Yaskawa INFORM job: SUPERDUPLEX_HALFBODY_11_02.JBI

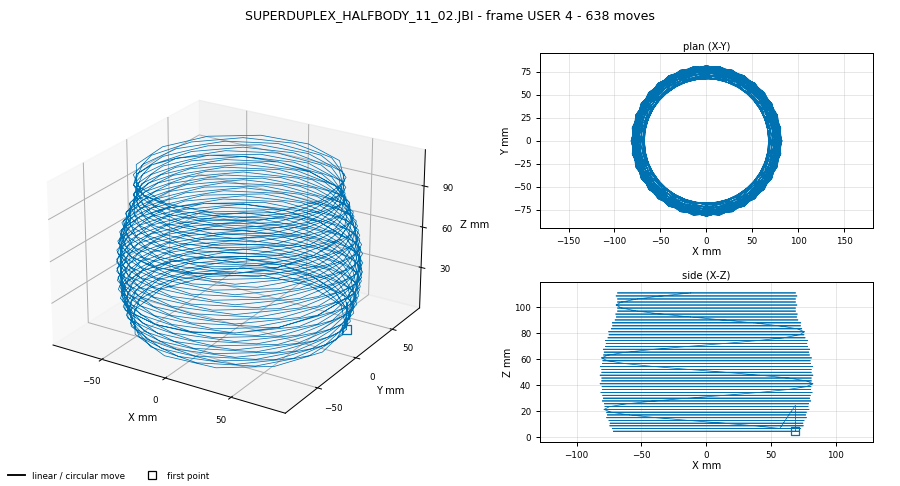
[picture p0: tool path of SUPERDUPLEX_HALFBODY_11_02.JBI in frame USER 4, 638 of 639 moves have a stored position in this frame; points joined in program order, loops and branches not executed]
/JOB
//NAME SUPERDUPLEX_HALFBODY_11_02
///FOLDERNAME SUPERDUPLEX_HALFBODY
//POS
///NPOS 638,0,639,1,0,0
///TOOL 9
///POSTYPE PULSE
P0=8353,-34220,-84194,-128214,7285,517082
///TOOL 9
///USER 4
///POSTYPE USER
///RECTAN
///RCONF 0,0,0,0,0,0,0,0,0,0,0,0,0,0,0,0,0,0,0,0,0,0,0,0
C0=68.785,24.654,4.486,-180.000,-180.000,134.719
C1=72.078,-12.983,4.486,-180.000,180.000,104.834
C2=56.111,-47.225,4.486,-180.000,180.000,74.949
C3=25.162,-68.896,4.486,-180.000,180.000,45.063
C4=-12.476,-72.189,4.486,180.000,180.000,15.136
C5=-46.717,-56.221,4.486,0.000,0.000,165.209
C6=-68.388,-25.273,4.486,0.000,0.000,135.282
C7=-71.681,12.365,4.486,0.000,0.000,105.166
C8=-55.714,46.607,4.486,0.000,0.000,75.051
C9=-24.765,68.278,4.486,0.000,0.000,44.936
C10=12.873,71.570,4.486,0.000,0.000,14.864
C11=47.115,55.603,4.486,-180.000,-180.000,164.791
C12=68.785,24.654,4.486,-180.000,-180.000,134.719
C13=68.785,24.654,24.486,-180.000,-180.000,134.719
C14=56.727,47.124,6.581,160.821,171.291,153.526
C15=25.437,69.033,6.581,-19.179,8.709,3.526
C16=-12.615,72.363,6.581,-19.179,8.709,33.526
C17=-47.234,56.219,6.581,-19.179,8.709,63.526
C18=-69.144,24.930,6.581,-19.179,8.709,93.526
C19=-72.473,-13.123,6.581,-19.179,8.709,123.526
C20=-56.330,-47.742,6.581,-19.179,8.709,153.526
C21=-25.040,-69.651,6.581,160.821,171.291,3.526
C22=13.013,-72.981,6.581,160.821,171.291,33.526
C23=47.632,-56.837,6.581,160.821,171.291,63.526
C24=69.541,-25.548,6.581,160.821,171.291,93.526
C25=72.870,12.505,6.581,160.821,171.291,123.526
C26=56.727,47.124,6.581,160.821,171.291,153.526
C27=37.536,64.360,8.629,158.693,170.383,173.187
C28=64.868,37.028,8.629,158.693,170.383,143.187
C29=74.872,-0.309,8.629,158.693,170.383,113.187
C30=64.868,-37.646,8.629,158.693,170.383,83.187
C31=37.536,-64.978,8.629,158.693,170.383,53.187
C32=0.199,-74.983,8.629,158.693,170.383,23.187
C33=-37.138,-64.978,8.629,-21.307,9.617,173.187
C34=-64.471,-37.646,8.629,-21.307,9.617,143.187
C35=-74.475,-0.309,8.629,-21.307,9.617,113.187
C36=-64.471,37.028,8.629,-21.307,9.617,83.187
C37=-37.138,64.360,8.629,-21.307,9.617,53.187
C38=0.199,74.365,8.629,-21.307,9.617,23.187
C39=37.536,64.360,8.629,158.693,170.383,173.187
C40=13.320,74.103,10.674,-21.438,9.672,13.165
C41=-25.644,70.694,10.674,-21.438,9.672,43.165
C42=-57.683,48.260,10.674,-21.438,9.672,73.165
C43=-74.213,12.812,10.674,-21.438,9.672,103.165
C44=-70.804,-26.152,10.674,-21.438,9.672,133.165
C45=-48.370,-58.191,10.674,-21.438,9.672,163.165
C46=-12.922,-74.721,10.674,158.562,170.328,13.165
C47=26.042,-71.312,10.674,158.562,170.328,43.165
C48=58.081,-48.878,10.674,158.562,170.328,73.165
C49=74.611,-13.430,10.674,158.562,170.328,103.165
C50=71.202,25.534,10.674,158.562,170.328,133.165
C51=48.768,57.573,10.674,158.562,170.328,163.165
C52=13.320,74.103,10.674,-21.438,9.672,13.165
C53=-13.072,74.951,12.739,-20.717,9.367,33.284
C54=26.336,71.504,12.739,-20.717,9.367,3.284
C55=58.741,48.814,12.739,159.283,170.633,153.284
C56=75.459,12.961,12.739,159.283,170.633,123.284
C57=72.012,-26.447,12.739,159.283,170.633,93.284
C58=49.322,-58.851,12.739,159.283,170.633,63.284
C59=13.469,-75.570,12.739,159.283,170.633,33.284
C60=-25.939,-72.122,12.739,159.283,170.633,3.284
C61=-58.344,-49.432,12.739,-20.717,9.367,153.284
C62=-75.062,-13.580,12.739,-20.717,9.367,123.284
C63=-71.614,25.829,12.739,-20.717,9.367,93.284
C64=-48.924,58.233,12.739,-20.717,9.367,63.284
C65=-13.072,74.951,12.739,-20.717,9.367,33.284
C66=-38.329,66.423,14.886,-14.976,6.871,54.096
C67=-66.533,38.219,14.886,-14.976,6.871,84.096
C68=-76.856,-0.309,14.886,-14.976,6.871,114.096
C69=-66.533,-38.837,14.886,-14.976,6.871,144.096
C70=-38.329,-67.041,14.886,-14.976,6.871,174.096
C71=0.199,-77.364,14.886,165.024,173.129,24.096
C72=38.726,-67.041,14.886,165.024,173.129,54.096
C73=66.931,-38.837,14.886,165.024,173.129,84.096
C74=77.254,-0.309,14.886,165.024,173.129,114.096
C75=66.931,38.219,14.886,165.024,173.129,144.096
C76=38.726,66.423,14.886,165.024,173.129,174.096
C77=0.199,76.746,14.886,-14.976,6.871,24.096
C78=-38.329,66.423,14.886,-14.976,6.871,54.096
C79=-59.325,49.637,17.023,-15.358,7.041,74.050
C80=-26.377,72.708,17.023,-15.358,7.041,44.050
C81=13.692,76.213,17.023,-15.358,7.041,14.050
C82=50.145,59.215,17.023,164.642,172.959,164.050
C83=73.216,26.267,17.023,164.642,172.959,134.050
C84=76.721,-13.802,17.023,164.642,172.959,104.050
C85=59.723,-50.256,17.023,164.642,172.959,74.049
C86=26.775,-73.326,17.023,164.642,172.959,44.050
C87=-13.294,-76.831,17.023,164.642,172.959,14.050
C88=-49.748,-59.833,17.023,-15.358,7.041,164.050
C89=-72.818,-26.885,17.023,-15.358,7.041,134.050
C90=-76.324,13.184,17.023,-15.358,7.041,104.050
C91=-59.325,49.637,17.023,-15.358,7.041,74.050
C92=-73.436,26.492,19.138,-15.733,7.206,94.003
C93=-76.971,-13.916,19.138,-15.733,7.206,124.003
C94=-59.829,-50.678,19.138,-15.733,7.206,154.003
C95=-26.602,-73.944,19.138,164.267,172.794,4.003
C96=13.806,-77.479,19.138,164.267,172.794,34.003
C97=50.568,-60.337,19.139,164.267,172.794,64.003
C98=73.834,-27.110,19.139,164.267,172.794,94.003
C99=77.369,13.298,19.139,164.267,172.794,124.003
C100=60.226,50.060,19.139,164.267,172.794,154.003
C101=27.000,73.326,19.139,-15.733,7.206,4.003
C102=-13.408,76.861,19.139,-15.733,7.206,34.003
C103=-50.170,59.719,19.139,-15.733,7.206,64.003
C104=-73.436,26.492,19.138,-15.733,7.206,94.003
C105=-78.847,-0.309,21.270,-16.233,7.427,113.939
C106=-68.256,39.214,21.270,-16.233,7.427,83.939
C107=-39.324,68.146,21.270,-16.233,7.427,53.939
C108=0.199,78.736,21.270,-16.233,7.427,23.939
C109=39.721,68.146,21.270,163.767,172.573,173.939
C110=68.654,39.214,21.270,163.767,172.573,143.939
C111=79.244,-0.309,21.270,163.767,172.573,113.939
C112=68.654,-39.832,21.270,163.767,172.573,83.939
C113=39.721,-68.764,21.270,163.767,172.573,53.939
C114=0.199,-79.354,21.270,163.767,172.573,23.939
C115=-39.324,-68.764,21.270,-16.233,7.427,173.939
C116=-68.256,-39.832,21.270,-16.233,7.427,143.939
C117=-78.847,-0.309,21.270,-16.233,7.427,113.939
C118=-74.567,-27.522,23.445,-12.204,5.630,134.398
C119=-50.944,-61.259,23.445,-12.204,5.630,164.398
C120=-13.617,-78.665,23.445,167.796,174.370,14.398
C121=27.411,-75.075,23.445,167.796,174.370,44.398
C122=61.149,-51.452,23.445,167.796,174.370,74.398
C123=78.554,-14.125,23.445,167.796,174.370,104.398
C124=74.965,26.904,23.445,167.796,174.370,134.398
C125=51.342,60.641,23.445,167.796,174.370,164.398
C126=14.015,78.047,23.445,-12.204,5.630,14.398
C127=-27.014,74.457,23.445,-12.204,5.630,44.398
C128=-60.751,50.834,23.445,-12.204,5.630,74.398
C129=-78.157,13.507,23.445,-12.204,5.630,104.398
C130=-74.567,-27.522,23.445,-12.204,5.630,134.398
C131=-61.063,-51.714,25.627,-9.595,4.444,154.627
C132=-78.558,-14.196,25.627,-9.595,4.444,124.627
C133=-74.950,27.043,25.627,-9.595,4.444,94.627
C134=-51.206,60.952,25.627,-9.595,4.444,64.627
C135=-13.688,78.447,25.627,-9.595,4.444,34.627
C136=27.551,74.839,25.627,-9.595,4.444,4.627
C137=61.460,51.095,25.627,170.405,175.556,154.627
C138=78.955,13.578,25.627,170.405,175.556,124.627
C139=75.347,-27.661,25.627,170.405,175.556,94.627
C140=51.603,-61.571,25.627,170.405,175.556,64.627
C141=14.086,-79.065,25.627,170.405,175.556,34.627
C142=-27.153,-75.457,25.627,170.405,175.556,4.627
C143=-61.063,-51.714,25.627,-9.595,4.444,154.627
C144=-39.992,-69.922,27.811,-9.673,4.480,174.621
C145=0.199,-80.691,27.811,170.327,175.520,24.621
C146=40.390,-69.922,27.811,170.327,175.520,54.621
C147=69.812,-40.500,27.811,170.327,175.520,84.621
C148=80.581,-0.309,27.811,170.327,175.520,114.621
C149=69.812,39.882,27.811,170.327,175.520,144.621
C150=40.390,69.304,27.811,170.327,175.520,174.621
C151=0.199,80.073,27.811,-9.673,4.480,24.621
C152=-39.992,69.304,27.811,-9.673,4.480,54.621
C153=-69.414,39.882,27.811,-9.673,4.480,84.621
C154=-80.183,-0.309,27.811,-9.673,4.480,114.621
C155=-69.414,-40.500,27.811,-9.673,4.480,144.621
C156=-39.992,-69.922,27.811,-9.673,4.480,174.621
C157=-13.839,-79.923,29.990,169.161,174.989,14.524
C158=-51.766,-62.238,29.990,-10.839,5.011,164.524
C159=-75.768,-27.959,29.990,-10.839,5.011,134.524
C160=-79.416,13.729,29.990,-10.839,5.011,104.524
C161=-61.730,51.655,29.990,-10.839,5.011,74.524
C162=-27.451,75.658,29.990,-10.839,5.011,44.524
C163=14.237,79.305,29.990,-10.839,5.011,14.524
C164=52.163,61.620,29.990,169.161,174.989,164.524
C165=76.166,27.341,29.990,169.161,174.989,134.524
C166=79.813,-14.347,29.990,169.161,174.989,104.524
C167=62.128,-52.274,29.990,169.161,174.989,74.524
C168=27.849,-76.276,29.990,169.161,174.989,44.524
C169=-13.839,-79.923,29.990,169.161,174.989,14.524
C170=14.319,-80.392,32.171,168.824,174.836,34.494
C171=52.469,-62.602,32.171,168.825,174.836,64.494
C172=76.613,-28.121,32.171,168.825,174.836,94.494
C173=80.281,13.812,32.171,168.825,174.836,124.494
C174=62.492,51.961,32.171,168.825,174.836,154.494
C175=28.011,76.105,32.171,-11.175,5.164,4.494
C176=-13.922,79.773,32.171,-11.175,5.164,34.494
C177=-52.071,61.984,32.171,-11.175,5.164,64.494
C178=-76.215,27.503,32.171,-11.176,5.164,94.494
C179=-79.884,-14.430,32.171,-11.176,5.164,124.494
C180=-62.094,-52.579,32.171,-11.176,5.164,154.494
C181=-27.614,-76.723,32.171,168.824,174.836,4.494
C182=14.319,-80.392,32.171,168.824,174.836,34.494
C183=40.929,-70.857,34.400,176.659,178.443,54.954
C184=0.199,-81.770,34.400,176.659,178.443,24.955
C185=-40.532,-70.857,34.400,-3.341,1.557,174.955
C186=-70.349,-41.040,34.400,-3.341,1.557,144.955
C187=-81.263,-0.309,34.400,-3.341,1.557,114.955
C188=-70.349,40.422,34.400,-3.341,1.557,84.955
C189=-40.532,70.239,34.400,-3.341,1.557,54.955
C190=0.199,81.152,34.400,-3.341,1.557,24.955
C191=40.929,70.239,34.400,176.659,178.443,174.955
C192=70.746,40.422,34.400,176.659,178.443,144.955
C193=81.660,-0.309,34.400,176.659,178.443,114.955
C194=70.746,-41.040,34.400,176.659,178.443,84.954
C195=40.929,-70.857,34.400,176.659,178.443,54.954
C196=62.746,-52.792,36.614,175.610,177.956,74.922
C197=80.607,-14.487,36.614,175.610,177.956,104.922
C198=76.924,27.617,36.614,175.610,177.956,134.922
C199=52.682,62.238,36.614,175.610,177.956,164.922
C200=14.377,80.100,36.614,-4.390,2.044,14.922
C201=-27.727,76.416,36.614,-4.390,2.044,44.922
C202=-62.348,52.174,36.614,-4.390,2.044,74.922
C203=-80.210,13.869,36.614,-4.390,2.044,104.922
C204=-76.526,-28.235,36.614,-4.390,2.044,134.922
C205=-52.284,-62.856,36.614,-4.390,2.044,164.922
C206=-13.979,-80.718,36.614,175.610,177.956,14.922
C207=28.124,-77.034,36.614,175.610,177.956,44.922
C208=62.746,-52.792,36.614,175.610,177.956,74.921
C209=77.111,-28.303,38.831,175.334,177.828,94.911
C210=52.810,-63.009,38.831,175.334,177.828,64.911
C211=14.412,-80.914,38.831,175.334,177.828,34.911
C212=-27.795,-77.222,38.831,175.334,177.828,4.911
C213=-62.501,-52.920,38.831,-4.666,2.172,154.912
C214=-80.406,-14.522,38.831,-4.666,2.172,124.912
C215=-76.714,27.685,38.831,-4.666,2.172,94.912
C216=-52.413,62.391,38.831,-4.666,2.172,64.912
C217=-14.014,80.296,38.831,-4.666,2.172,34.912
C218=28.193,76.604,38.831,-4.666,2.172,4.912
C219=62.898,52.302,38.831,175.334,177.828,154.912
C220=80.804,13.904,38.831,175.334,177.828,124.911
C221=77.111,-28.303,38.831,175.334,177.828,94.911
C222=82.288,-0.309,41.051,174.396,177.393,114.872
C223=71.290,40.735,41.051,174.396,177.393,144.872
C224=41.243,70.782,41.051,174.396,177.393,174.872
C225=0.199,81.780,41.051,-5.604,2.607,24.872
C226=-40.846,70.782,41.051,-5.604,2.607,54.872
C227=-70.892,40.735,41.051,-5.604,2.607,84.872
C228=-81.890,-0.309,41.051,-5.604,2.607,114.872
C229=-70.892,-41.354,41.051,-5.604,2.607,144.872
C230=-40.846,-71.400,41.051,-5.604,2.607,174.872
C231=0.199,-82.398,41.051,174.396,177.393,24.872
C232=41.243,-71.400,41.051,174.396,177.393,54.872
C233=71.290,-41.354,41.051,174.396,177.393,84.872
C234=82.288,-0.309,41.051,174.396,177.393,114.872
C235=77.438,27.804,43.278,177.496,178.833,134.974
C236=81.146,-14.582,43.278,177.496,178.833,104.974
C237=63.165,-53.144,43.278,177.496,178.833,74.974
C238=28.312,-77.548,43.278,177.496,178.833,44.974
C239=-14.075,-81.257,43.278,177.496,178.833,14.974
C240=-52.636,-63.275,43.278,-2.504,1.167,164.974
C241=-77.041,-28.422,43.278,-2.504,1.167,134.975
C242=-80.749,13.964,43.278,-2.504,1.167,104.975
C243=-62.767,52.526,43.278,-2.504,1.167,74.975
C244=-27.914,76.930,43.278,-2.504,1.167,44.975
C245=14.472,80.639,43.278,-2.504,1.167,14.975
C246=53.034,62.657,43.278,177.496,178.833,164.975
C247=77.438,27.804,43.278,177.496,178.833,134.974
C248=63.104,52.474,45.501,-178.135,-179.131,154.986
C249=28.284,76.855,45.501,1.865,-0.869,4.986
C250=-14.061,80.560,45.501,1.865,-0.869,34.986
C251=-52.585,62.596,45.501,1.865,-0.869,64.986
C252=-76.966,27.776,45.501,1.865,-0.869,94.986
C253=-80.670,-14.568,45.501,1.865,-0.869,124.986
C254=-62.706,-53.093,45.501,1.865,-0.869,154.986
C255=-27.887,-77.473,45.501,-178.135,-179.131,4.986
C256=14.458,-81.178,45.501,-178.135,-179.131,34.986
C257=52.982,-63.214,45.501,-178.135,-179.131,64.986
C258=77.363,-28.395,45.501,-178.135,-179.131,94.986
C259=81.068,13.950,45.501,-178.135,-179.131,124.986
C260=63.104,52.474,45.501,-178.135,-179.131,154.986
C261=41.238,70.773,47.716,-179.117,-179.588,174.997
C262=71.281,40.730,47.716,-179.117,-179.588,144.997
C263=82.278,-0.309,47.716,-179.117,-179.588,114.997
C264=71.281,-41.348,47.716,-179.117,-179.588,84.997
C265=41.238,-71.391,47.716,-179.117,-179.588,54.997
C266=0.199,-82.388,47.716,-179.117,-179.588,24.997
C267=-40.841,-71.391,47.716,0.883,-0.412,174.997
C268=-70.884,-41.348,47.716,0.883,-0.412,144.997
C269=-81.880,-0.309,47.716,0.883,-0.412,114.997
C270=-70.884,40.730,47.716,0.883,-0.412,84.996
C271=-40.841,70.773,47.716,0.883,-0.412,54.996
C272=0.199,81.770,47.716,0.883,-0.412,24.997
C273=41.238,70.773,47.716,-179.117,-179.588,174.997
C274=14.448,80.500,49.940,0.540,-0.250,14.824
C275=-27.866,76.798,49.940,0.540,-0.251,44.945
C276=-62.660,52.435,49.940,0.539,-0.252,75.067
C277=-80.610,13.940,49.940,0.538,-0.253,105.188
C278=-76.908,-28.374,49.940,0.538,-0.253,135.183
C279=-52.546,-63.167,49.940,0.539,-0.253,165.178
C280=-14.050,-81.118,49.940,-179.461,-179.747,15.172
C281=28.263,-77.416,49.940,-179.461,-179.748,45.052
C282=63.057,-53.053,49.940,-179.460,-179.749,74.931
C283=81.008,-14.558,49.940,-179.460,-179.750,104.811
C284=77.306,27.756,49.940,-179.460,-179.750,134.815
C285=52.943,62.549,49.940,-179.460,-179.750,164.820
C286=14.448,80.500,49.940,0.540,-0.250,14.824
C287=-14.047,80.481,52.179,0.444,-0.206,34.900
C288=28.257,76.780,52.179,0.444,-0.206,4.854
C289=63.042,52.423,52.179,-179.556,-179.795,154.808
C290=80.989,13.936,52.179,-179.555,-179.795,124.763
C291=77.288,-28.367,52.179,-179.556,-179.794,94.875
C292=52.931,-63.153,52.179,-179.556,-179.793,64.986
C293=14.444,-81.099,52.179,-179.557,-179.792,35.098
C294=-27.859,-77.398,52.179,-179.557,-179.792,5.144
C295=-62.645,-53.041,52.179,0.443,-0.208,155.190
C296=-80.592,-14.555,52.179,0.443,-0.209,125.236
C297=-76.890,27.749,52.179,0.443,-0.208,95.124
C298=-52.533,62.535,52.179,0.444,-0.207,65.012
C299=-14.047,80.481,52.179,0.444,-0.206,34.900
C300=-40.705,70.538,54.403,5.357,-2.493,54.883
C301=-70.648,40.594,54.403,5.357,-2.493,84.883
C302=-81.608,-0.309,54.403,5.357,-2.493,114.883
C303=-70.648,-41.212,54.403,5.357,-2.493,144.883
C304=-40.705,-71.156,54.403,5.357,-2.493,174.883
C305=0.199,-82.116,54.403,-174.643,-177.507,24.883
C306=41.102,-71.156,54.403,-174.643,-177.507,54.883
C307=71.045,-41.212,54.403,-174.643,-177.507,84.883
C308=82.005,-0.309,54.403,-174.643,-177.507,114.883
C309=71.045,40.594,54.403,-174.643,-177.507,144.883
C310=41.102,70.538,54.403,-174.643,-177.507,174.883
C311=0.199,81.498,54.403,5.357,-2.493,24.883
C312=-40.705,70.538,54.403,5.357,-2.493,54.883
C313=-62.243,52.086,56.608,6.895,-3.204,74.807
C314=-27.680,76.287,56.608,6.895,-3.204,44.807
C315=14.353,79.965,56.608,6.895,-3.204,14.807
C316=52.594,62.133,56.608,-173.105,-176.796,164.807
C317=76.795,27.570,56.608,-173.105,-176.796,134.807
C318=80.473,-14.464,56.608,-173.105,-176.796,104.807
C319=62.641,-52.704,56.608,-173.105,-176.796,74.807
C320=28.078,-76.906,56.608,-173.105,-176.796,44.807
C321=-13.956,-80.583,56.608,-173.105,-176.796,14.807
C322=-52.196,-62.751,56.608,6.895,-3.204,164.807
C323=-76.398,-28.188,56.608,6.895,-3.204,134.807
C324=-80.075,13.845,56.608,6.895,-3.204,104.807
C325=-62.243,52.086,56.608,6.895,-3.204,74.807
C326=-76.156,27.482,58.803,6.073,-2.824,94.850
C327=-79.821,-14.419,58.803,6.073,-2.824,124.850
C328=-62.046,-52.539,58.803,6.073,-2.824,154.850
C329=-27.592,-76.663,58.803,-173.927,-177.176,4.850
C330=14.308,-80.329,58.803,-173.927,-177.176,34.850
C331=52.428,-62.554,58.803,-173.927,-177.176,64.850
C332=76.553,-28.100,58.803,-173.927,-177.176,94.850
C333=80.219,13.801,58.803,-173.927,-177.176,124.850
C334=62.443,51.920,58.803,-173.927,-177.176,154.850
C335=27.989,76.045,58.803,6.073,-2.824,4.850
C336=-13.911,79.711,58.803,6.073,-2.824,34.850
C337=-52.031,61.936,58.803,6.073,-2.824,64.850
C338=-76.156,27.482,58.803,6.073,-2.824,94.850
C339=-80.810,-0.309,61.018,5.751,-2.675,114.866
C340=-69.957,40.195,61.018,5.751,-2.675,84.866
C341=-40.305,69.846,61.018,5.751,-2.675,54.866
C342=0.199,80.699,61.018,5.751,-2.675,24.866
C343=40.703,69.846,61.018,-174.249,-177.325,174.866
C344=70.354,40.195,61.018,-174.249,-177.325,144.866
C345=81.207,-0.309,61.018,-174.249,-177.325,114.866
C346=70.354,-40.813,61.018,-174.249,-177.325,84.866
C347=40.703,-70.464,61.018,-174.249,-177.325,54.866
C348=0.199,-81.318,61.018,-174.249,-177.325,24.866
C349=-40.305,-70.464,61.018,5.751,-2.675,174.866
C350=-69.957,-40.813,61.018,5.751,-2.675,144.866
C351=-80.810,-0.309,61.018,5.751,-2.675,114.866
C352=-75.629,-27.908,63.281,7.174,-3.333,134.791
C353=-51.670,-62.124,63.281,7.174,-3.333,164.791
C354=-13.814,-79.777,63.281,-172.826,-176.667,14.791
C355=27.798,-76.137,63.281,-172.826,-176.667,44.791
C356=62.014,-52.178,63.281,-172.826,-176.667,74.791
C357=79.667,-14.321,63.281,-172.826,-176.667,104.791
C358=76.026,27.290,63.281,-172.826,-176.667,134.791
C359=52.068,61.506,63.281,-172.826,-176.667,164.791
C360=14.211,79.159,63.281,7.174,-3.333,14.791
C361=-27.400,75.519,63.281,7.174,-3.333,44.791
C362=-61.617,51.560,63.281,7.174,-3.333,74.791
C363=-79.270,13.703,63.281,7.174,-3.333,104.791
C364=-75.629,-27.908,63.281,7.174,-3.333,134.791
C365=-61.206,-51.834,65.507,12.309,-5.677,154.387
C366=-78.742,-14.228,65.507,12.309,-5.677,124.387
C367=-75.125,27.107,65.507,12.309,-5.677,94.387
C368=-51.326,61.096,65.507,12.309,-5.677,64.387
C369=-13.721,78.632,65.507,12.309,-5.677,34.387
C370=27.615,75.015,65.507,12.309,-5.677,4.387
C371=61.604,51.216,65.507,-167.691,-174.323,154.387
C372=79.139,13.610,65.507,-167.691,-174.323,124.387
C373=75.523,-27.725,65.507,-167.691,-174.323,94.387
C374=51.724,-61.714,65.507,-167.691,-174.323,64.387
C375=14.118,-79.250,65.507,-167.691,-174.323,34.387
C376=-27.217,-75.633,65.507,-167.691,-174.323,4.387
C377=-61.206,-51.834,65.507,12.309,-5.677,154.387
C378=-39.615,-69.269,67.708,12.315,-5.680,174.387
C379=0.199,-79.937,67.709,-167.685,-174.320,24.387
C380=40.013,-69.269,67.709,-167.685,-174.320,54.387
C381=69.159,-40.123,67.709,-167.685,-174.320,84.387
C382=79.827,-0.309,67.709,-167.685,-174.320,114.387
C383=69.159,39.505,67.709,-167.685,-174.320,144.387
C384=40.013,68.651,67.709,-167.685,-174.320,174.387
C385=0.199,79.319,67.709,12.315,-5.680,24.387
C386=-39.615,68.651,67.709,12.315,-5.680,54.387
C387=-68.761,39.505,67.709,12.315,-5.680,84.387
C388=-79.429,-0.309,67.709,12.315,-5.680,114.387
C389=-68.761,-40.123,67.708,12.315,-5.680,144.387
C390=-39.615,-69.269,67.708,12.315,-5.680,174.387
C391=-13.542,-78.238,69.931,-168.546,-174.709,14.469
C392=-50.666,-60.927,69.931,11.454,-5.291,164.469
C393=-74.160,-27.374,69.931,11.454,-5.291,134.469
C394=-77.730,13.432,69.931,11.454,-5.291,104.469
C395=-60.419,50.555,69.931,11.454,-5.291,74.469
C396=-26.866,74.050,69.931,11.454,-5.291,44.469
C397=13.940,77.620,69.931,11.454,-5.291,14.469
C398=51.063,60.309,69.931,-168.546,-174.709,164.469
C399=74.558,26.755,69.931,-168.546,-174.709,134.469
C400=78.128,-14.050,69.931,-168.546,-174.709,104.469
C401=60.817,-51.174,69.931,-168.546,-174.709,74.469
C402=27.263,-74.668,69.931,-168.546,-174.709,44.469
C403=-13.542,-78.238,69.931,-168.546,-174.709,14.469
C404=13.847,-77.714,72.142,-167.688,-174.321,34.387
C405=50.721,-60.519,72.142,-167.688,-174.321,64.387
C406=74.057,-27.191,72.142,-167.688,-174.321,94.387
C407=77.603,13.339,72.142,-167.688,-174.321,124.387
C408=60.409,50.213,72.142,-167.688,-174.321,154.387
C409=27.081,73.550,72.142,12.312,-5.679,4.387
C410=-13.450,77.096,72.142,12.312,-5.679,34.387
C411=-50.323,59.901,72.142,12.312,-5.679,64.387
C412=-73.660,26.573,72.142,12.312,-5.679,94.387
C413=-77.206,-13.958,72.142,12.312,-5.679,124.387
C414=-60.011,-50.831,72.142,12.312,-5.679,154.387
C415=-26.684,-74.168,72.142,-167.688,-174.321,4.387
C416=13.847,-77.714,72.142,-167.688,-174.321,34.387
C417=39.200,-67.861,74.351,-166.249,-173.675,54.237
C418=0.199,-78.311,74.351,-166.249,-173.675,24.237
C419=-38.802,-67.861,74.351,13.751,-6.325,174.237
C420=-67.353,-39.310,74.351,13.751,-6.325,144.237
C421=-77.804,-0.309,74.351,13.751,-6.325,114.237
C422=-67.353,38.692,74.351,13.751,-6.325,84.237
C423=-38.802,67.243,74.351,13.751,-6.325,54.236
C424=0.199,77.693,74.351,13.751,-6.325,24.237
C425=39.200,67.243,74.351,-166.249,-173.675,174.237
C426=67.751,38.692,74.351,-166.249,-173.675,144.237
C427=78.201,-0.309,74.351,-166.249,-173.675,114.237
C428=67.751,-39.310,74.351,-166.249,-173.675,84.237
C429=39.200,-67.861,74.351,-166.249,-173.675,54.237
C430=59.364,-49.955,76.505,-162.106,-171.846,73.714
C431=76.260,-13.721,76.505,-162.106,-171.846,103.714
C432=72.776,26.107,76.505,-162.106,-171.846,133.714
C433=49.844,58.856,76.505,-162.106,-171.846,163.714
C434=13.610,75.752,76.505,17.894,-8.154,13.714
C435=-26.217,72.268,76.505,17.894,-8.154,43.714
C436=-58.967,49.337,76.505,17.894,-8.154,73.714
C437=-75.863,13.103,76.505,17.894,-8.154,103.714
C438=-72.378,-26.725,76.505,17.894,-8.154,133.714
C439=-49.447,-59.474,76.505,17.894,-8.154,163.714
C440=-13.213,-76.371,76.505,-162.106,-171.846,13.714
C441=26.615,-72.886,76.505,-162.106,-171.846,43.714
C442=59.364,-49.955,76.505,-162.106,-171.846,73.714
C443=71.980,-26.435,78.831,-161.742,-171.688,93.662
C444=49.300,-58.826,78.831,-161.742,-171.688,63.662
C445=13.463,-75.537,78.831,-161.742,-171.688,33.662
C446=-25.928,-72.090,78.831,-161.742,-171.688,3.662
C447=-58.318,-49.410,78.831,18.258,-8.312,153.662
C448=-75.029,-13.574,78.831,18.258,-8.312,123.662
C449=-71.583,25.817,78.831,18.258,-8.312,93.662
C450=-48.903,58.208,78.831,18.258,-8.312,63.662
C451=-13.066,74.919,78.831,18.258,-8.312,33.662
C452=26.325,71.472,78.831,18.258,-8.312,3.662
C453=58.715,48.792,78.831,-161.742,-171.688,153.662
C454=75.426,12.956,78.831,-161.742,-171.688,123.662
C455=71.980,-26.435,78.831,-161.742,-171.688,93.662
C456=75.712,-0.309,81.150,-161.130,-171.424,113.572
C457=65.595,37.448,81.150,-161.130,-171.424,143.572
C458=37.955,65.087,81.150,-161.130,-171.424,173.572
C459=0.199,75.204,81.150,18.870,-8.576,23.572
C460=-37.558,65.087,81.150,18.870,-8.576,53.572
C461=-65.198,37.448,81.150,18.870,-8.576,83.572
C462=-75.315,-0.309,81.150,18.870,-8.576,113.572
C463=-65.198,-38.066,81.150,18.870,-8.576,143.572
C464=-37.558,-65.706,81.150,18.870,-8.576,173.572
C465=0.199,-75.822,81.150,-161.130,-171.424,23.572
C466=37.955,-65.706,81.150,-161.130,-171.424,53.572
C467=65.595,-38.066,81.150,-161.130,-171.424,83.572
C468=75.712,-0.309,81.150,-161.130,-171.424,113.572
C469=70.309,25.209,83.460,-160.464,-171.137,133.471
C470=73.675,-13.265,83.460,-160.464,-171.137,103.471
C471=57.353,-48.267,83.460,-160.464,-171.137,73.471
C472=25.717,-70.419,83.460,-160.464,-171.137,43.471
C473=-12.757,-73.785,83.460,-160.464,-171.137,13.471
C474=-47.759,-57.463,83.460,19.536,-8.863,163.471
C475=-69.911,-25.827,83.460,19.536,-8.863,133.471
C476=-73.277,12.647,83.460,19.536,-8.863,103.471
C477=-56.955,47.649,83.460,19.536,-8.863,73.471
C478=-25.319,69.801,83.460,19.536,-8.863,43.471
C479=13.155,73.167,83.460,19.536,-8.863,13.471
C480=48.157,56.845,83.460,-160.464,-171.137,163.471
C481=70.309,25.209,83.460,-160.464,-171.137,133.471
C482=56.619,47.033,85.745,-159.192,-170.594,153.269
C483=25.389,68.900,85.745,20.808,-9.406,3.269
C484=-12.591,72.223,85.745,20.808,-9.406,33.269
C485=-47.143,56.111,85.745,20.808,-9.406,63.269
C486=-69.011,24.881,85.745,20.808,-9.406,93.269
C487=-72.333,-13.098,85.745,20.808,-9.406,123.269
C488=-56.221,-47.651,85.745,20.808,-9.406,153.269
C489=-24.991,-69.518,85.745,-159.192,-170.594,3.269
C490=12.988,-72.841,85.745,-159.192,-170.594,33.269
C491=47.541,-56.729,85.745,-159.192,-170.594,63.269
C492=69.408,-25.499,85.745,-159.192,-170.594,93.269
C493=72.731,12.480,85.745,-159.192,-170.594,123.269
C494=56.619,47.033,85.745,-159.192,-170.594,153.269
C495=36.548,62.649,88.043,-159.395,-170.681,173.302
C496=63.157,36.040,88.043,-159.395,-170.681,143.302
C497=72.897,-0.309,88.043,-159.395,-170.681,113.302
C498=63.157,-36.658,88.043,-159.395,-170.681,83.302
C499=36.548,-63.267,88.043,-159.395,-170.681,53.302
C500=0.199,-73.007,88.043,-159.395,-170.681,23.302
C501=-36.150,-63.267,88.043,20.605,-9.319,173.302
C502=-62.760,-36.658,88.043,20.605,-9.319,143.302
C503=-72.499,-0.309,88.043,20.605,-9.319,113.302
C504=-62.760,36.040,88.043,20.605,-9.319,83.302
C505=-36.150,62.649,88.043,20.605,-9.319,53.302
C506=0.199,72.389,88.043,20.605,-9.319,23.302
C507=36.548,62.649,88.043,-159.395,-170.681,173.302
C508=12.633,70.212,90.292,23.699,-10.616,12.767
C509=-24.293,66.981,90.292,23.699,-10.616,42.767
C510=-54.657,45.720,90.292,23.699,-10.616,72.767
C511=-70.322,12.126,90.292,23.699,-10.616,102.767
C512=-67.091,-24.801,90.292,23.699,-10.616,132.767
C513=-45.830,-55.164,90.292,23.699,-10.616,162.767
C514=-12.236,-70.830,90.292,-156.301,-169.384,12.767
C515=24.690,-67.599,90.292,-156.301,-169.384,42.767
C516=55.054,-46.338,90.292,-156.301,-169.384,72.767
C517=70.719,-12.744,90.292,-156.301,-169.384,102.767
C518=67.489,24.183,90.292,-156.301,-169.384,132.767
C519=46.228,54.546,90.292,-156.301,-169.384,162.767
C520=12.633,70.212,90.292,23.699,-10.616,12.767
C521=-12.069,69.262,92.596,20.771,-9.390,33.275
C522=24.361,66.075,92.596,20.771,-9.390,3.275
C523=54.315,45.100,92.596,-159.229,-170.610,153.275
C524=69.770,11.958,92.596,-159.229,-170.610,123.275
C525=66.583,-24.471,92.596,-159.229,-170.610,93.275
C526=45.608,-54.426,92.596,-159.229,-170.610,63.275
C527=12.466,-69.880,92.596,-159.229,-170.610,33.275
C528=-23.963,-66.693,92.596,-159.229,-170.610,3.275
C529=-53.918,-45.718,92.596,20.771,-9.390,153.275
C530=-69.372,-12.576,92.596,20.771,-9.390,123.275
C531=-66.185,23.853,92.596,20.771,-9.390,93.275
C532=-45.211,53.808,92.596,20.771,-9.390,63.275
C533=-12.069,69.262,92.596,20.771,-9.390,33.275
C534=-34.828,60.358,94.847,13.396,-6.166,54.275
C535=-60.469,34.717,94.847,13.396,-6.166,84.275
C536=-69.854,-0.309,94.847,13.396,-6.166,114.275
C537=-60.469,-35.335,94.847,13.396,-6.166,144.275
C538=-34.828,-60.976,94.847,13.396,-6.166,174.275
C539=0.199,-70.362,94.847,-166.604,-173.834,24.275
C540=35.225,-60.976,94.847,-166.604,-173.834,54.275
C541=60.866,-35.335,94.847,-166.604,-173.834,84.275
C542=70.251,-0.309,94.847,-166.604,-173.834,114.275
C543=60.866,34.717,94.847,-166.604,-173.834,144.275
C544=35.225,60.358,94.847,-166.604,-173.834,174.275
C545=0.199,69.744,94.847,13.396,-6.166,24.275
C546=-34.828,60.358,94.847,13.396,-6.166,54.275
C547=-53.252,44.542,97.159,6.209,-2.887,74.843
C548=-23.666,65.258,97.159,6.209,-2.887,44.843
C549=12.315,68.406,97.159,6.209,-2.887,14.843
C550=45.049,53.142,97.159,-173.791,-177.113,164.843
C551=65.766,23.555,97.159,-173.791,-177.113,134.843
C552=68.914,-12.425,97.159,-173.791,-177.113,104.843
C553=53.650,-45.160,97.159,-173.791,-177.113,74.843
C554=24.063,-65.876,97.159,-173.791,-177.113,44.843
C555=-11.918,-69.024,97.159,-173.791,-177.113,14.843
C556=-44.652,-53.760,97.159,6.209,-2.887,164.843
C557=-65.368,-24.174,97.159,6.209,-2.887,134.843
C558=-68.516,11.807,97.159,6.209,-2.887,104.843
C559=-53.252,44.542,97.159,6.209,-2.887,74.843
C560=-65.341,23.545,99.489,0.650,-0.306,95.182
C561=-68.488,-12.420,99.489,0.650,-0.306,125.200
C562=-53.230,-45.141,99.489,0.650,-0.306,155.219
C563=-23.656,-65.849,99.489,-179.351,-179.694,5.238
C564=12.310,-68.995,99.489,-179.350,-179.695,35.097
C565=45.031,-53.738,99.489,-179.349,-179.697,64.957
C566=65.739,-24.164,99.489,-179.348,-179.699,94.816
C567=68.885,11.802,99.489,-179.348,-179.699,124.797
C568=53.627,44.523,99.489,-179.348,-179.699,154.777
C569=24.053,65.231,99.489,0.652,-0.301,4.757
C570=-11.913,68.377,99.489,0.651,-0.302,34.899
C571=-44.633,53.119,99.489,0.650,-0.304,65.040
C572=-65.341,23.545,99.489,0.650,-0.306,95.182
C573=-69.543,-0.309,101.819,0.089,-0.042,115.255
C574=-60.200,34.562,101.819,0.090,-0.042,85.115
C575=-34.672,60.089,101.819,0.090,-0.042,54.976
C576=0.199,69.433,101.819,0.090,-0.042,24.836
C577=35.070,60.089,101.819,-179.910,-179.959,174.806
C578=60.597,34.562,101.819,-179.910,-179.959,144.777
C579=69.941,-0.309,101.819,-179.910,-179.959,114.747
C580=60.597,-35.180,101.819,-179.910,-179.958,84.885
C581=35.070,-60.707,101.819,-179.910,-179.958,55.024
C582=0.199,-70.051,101.819,-179.911,-179.958,25.163
C583=-34.672,-60.707,101.819,0.089,-0.042,175.193
C584=-60.200,-35.180,101.819,0.089,-0.042,145.224
C585=-69.543,-0.309,101.819,0.089,-0.042,115.255
C586=-65.336,-24.162,104.149,0.025,-0.012,135.295
C587=-44.630,-53.734,104.149,0.025,-0.012,165.219
C588=-11.912,-68.990,104.149,-179.975,-179.988,15.142
C589=24.052,-65.844,104.149,-179.975,-179.989,45.066
C590=53.623,-45.138,104.149,-179.975,-179.989,74.946
C591=68.880,-12.419,104.149,-179.975,-179.989,104.826
C592=65.734,23.544,104.149,-179.975,-179.989,134.706
C593=45.027,53.116,104.149,-179.975,-179.989,164.782
C594=12.309,68.372,104.149,0.025,-0.011,14.857
C595=-23.654,65.226,104.149,0.025,-0.011,44.933
C596=-53.226,44.520,104.149,0.025,-0.011,75.054
C597=-68.483,11.801,104.149,0.025,-0.012,105.174
C598=-65.336,-24.162,104.149,0.025,-0.012,135.295
C599=-53.227,-45.139,106.479,-0.039,0.019,155.299
C600=-68.484,-12.420,106.479,-0.039,0.018,125.212
C601=-65.338,23.544,106.479,-0.039,0.018,95.125
C602=-44.631,53.117,106.479,-0.039,0.018,65.038
C603=-11.912,68.374,106.479,-0.039,0.018,34.926
C604=24.052,65.228,106.479,-0.039,0.018,4.813
C605=53.625,44.521,106.479,179.961,179.982,154.700
C606=68.882,11.802,106.479,179.961,179.982,124.788
C607=65.735,-24.162,106.479,179.961,179.982,94.875
C608=45.028,-53.735,106.479,179.961,179.982,64.962
C609=12.309,-68.992,106.479,179.961,179.982,35.074
C610=-23.655,-65.846,106.479,179.961,179.982,5.187
C611=-53.227,-45.139,106.479,-0.039,0.019,155.299
C612=-34.675,-60.712,108.809,-0.103,0.049,175.268
C613=0.199,-70.056,108.809,179.897,179.951,25.133
C614=35.072,-60.712,108.809,179.897,179.952,54.997
C615=60.602,-35.183,108.809,179.896,179.952,84.862
C616=69.946,-0.309,108.809,179.896,179.952,114.819
C617=60.602,34.565,108.809,179.896,179.952,144.775
C618=35.072,60.094,108.809,179.896,179.952,174.731
C619=0.199,69.438,108.809,-0.104,0.048,24.867
C620=-34.675,60.094,108.809,-0.103,0.048,55.003
C621=-60.204,34.565,108.809,-0.103,0.048,85.139
C622=-69.549,-0.309,108.809,-0.103,0.049,115.182
C623=-60.204,-35.183,108.809,-0.103,0.049,145.225
C624=-34.675,-60.712,108.809,-0.103,0.049,175.268
C625=-11.914,-69.003,111.139,179.865,179.936,15.204
C626=-44.638,-53.743,111.138,-0.135,0.064,165.210
C627=-65.348,-24.166,111.138,-0.135,0.064,135.216
C628=-68.495,11.803,111.139,-0.135,0.064,105.222
C629=-53.235,44.528,111.139,-0.135,0.063,75.080
C630=-23.658,65.238,111.139,-0.135,0.063,44.937
C631=12.311,68.385,111.139,-0.135,0.063,14.794
C632=45.035,53.125,111.139,179.865,179.937,164.789
C633=65.745,23.548,111.139,179.865,179.937,134.784
C634=68.892,-12.422,111.139,179.865,179.937,104.779
C635=53.633,-45.146,111.139,179.865,179.937,74.921
C636=24.056,-65.856,111.139,179.865,179.937,45.062
C637=-11.914,-69.003,111.139,179.865,179.936,15.204
///TOOL 0
///POSTYPE PULSE
///PULSE
EC0=-1624.2458,225496.6318
EC1=-1624.2458,225496.6318
EC2=-1624.2319,321383.3629
EC3=-1624.2179,417270.0939
EC4=-1624.2039,513156.8250
EC5=-1624.1983,609178.3288
EC6=-1624.1926,705199.8327
EC7=-1624.1869,801221.3365
EC8=-1624.2010,897845.9680
EC9=-1624.2150,994470.5996
EC10=-1624.2290,1091095.2312
EC11=-1624.2346,1187582.3566
EC12=-1624.2402,1284069.4819
EC13=-1624.2458,1380556.6073
EC14=-1624.2458,1380556.6073
EC15=65740.5181,1315485.0000
EC16=65740.5283,1219229.9674
EC17=65740.5385,1122974.9347
EC18=65740.5487,1026719.9021
EC19=65740.5609,930464.9347
EC20=65740.5731,834209.9674
EC21=65740.5854,737955.0000
EC22=65740.5752,641700.0326
EC23=65740.5650,545445.0653
EC24=65740.5548,449190.0979
EC25=65740.5425,352935.0653
EC26=65740.5303,256680.0326
EC27=65740.5181,160425.0000
EC28=73083.5982,96254.9755
EC29=73083.6043,192510.0082
EC30=73083.6104,288765.0408
EC31=73083.6165,385020.0734
EC32=73083.6308,481275.0490
EC33=73083.6451,577530.0245
EC34=73083.6593,673785.0000
EC35=73083.6512,770039.9674
EC36=73083.6430,866294.9347
EC37=73083.6349,962549.9021
EC38=73083.6226,1058804.9347
EC39=73083.6104,1155059.9674
EC40=73083.5982,1251315.0000
EC41=73535.6931,1187145.0000
EC42=73535.7073,1090889.9674
EC43=73535.7216,994634.9347
EC44=73535.7359,898379.9021
EC45=73535.7379,802124.9510
EC46=73535.7400,705870.0000
EC47=73535.7420,609615.0490
EC48=73535.7298,513360.0490
EC49=73535.7175,417105.0490
EC50=73535.7053,320850.0490
EC51=73535.7012,224595.0163
EC52=73535.6971,128339.9837
EC53=73535.6931,32084.9510
EC54=71051.1324,-32085.0673
EC55=71051.1304,64169.9714
EC56=71051.1283,160425.0102
EC57=71051.1263,256680.0490
EC58=71051.1426,352935.0490
EC59=71051.1589,449190.0490
EC60=71051.1753,545445.0490
EC61=71051.1793,641700.0326
EC62=71051.1834,737955.0163
EC63=71051.1875,834210.0000
EC64=71051.1691,930464.9674
EC65=71051.1508,1026719.9347
EC66=71051.1324,1122974.9021
EC67=51137.0385,1058804.9021
EC68=51137.0527,962549.9184
EC69=51137.0670,866294.9347
EC70=51137.0813,770039.9510
EC71=51137.0731,673785.0000
EC72=51137.0650,577530.0490
EC73=51137.0568,481275.0979
EC74=51137.0436,385020.0734
EC75=51137.0303,288765.0490
EC76=51137.0170,192510.0245
EC77=51137.0242,96254.9796
EC78=51137.0313,-0.0653
EC79=51137.0385,-96255.1102
EC80=52470.0958,-160425.1102
EC81=52470.0835,-64170.0775
EC82=52470.0713,32084.9551
EC83=52470.0591,128339.9878
EC84=52470.0693,224595.0245
EC85=52470.0795,320850.0612
EC86=52470.0897,417105.0979
EC87=52470.1019,513360.0653
EC88=52470.1141,609615.0326
EC89=52470.1264,705870.0000
EC90=52470.1162,802124.9674
EC91=52470.1060,898379.9347
EC92=52470.0958,994634.9021
EC93=53777.1595,930464.9021
EC94=53777.1636,834209.9510
EC95=53777.1677,737955.0000
EC96=53777.1718,641700.0490
EC97=53777.1575,545445.0653
EC98=53777.1432,449190.0816
EC99=53777.1289,352935.0979
EC100=53777.1249,256680.0490
EC101=53777.1208,160425.0000
EC102=53777.1167,64169.9510
EC103=53777.1310,-32085.0653
EC104=53777.1453,-128340.0816
EC105=53777.1595,-224595.0979
EC106=55519.6726,-288765.0734
EC107=55519.6562,-192510.0490
EC108=55519.6399,-96255.0245
EC109=55519.6236,0.0000
EC110=55519.6256,96255.0245
EC111=55519.6277,192510.0490
EC112=55519.6297,288765.0734
EC113=55519.6440,385020.0490
EC114=55519.6583,481275.0245
EC115=55519.6726,577530.0000
EC116=55519.6726,673784.9674
EC117=55519.6726,770039.9347
EC118=55519.6726,866294.9021
EC119=41440.0570,802124.9510
EC120=41440.0519,705870.0000
EC121=41440.0468,609615.0490
EC122=41440.0417,513360.0979
EC123=41440.0274,417105.0816
EC124=41440.0131,320850.0653
EC125=41439.9988,224595.0490
EC126=41440.0050,128339.9898
EC127=41440.0111,32084.9306
EC128=41440.0172,-64170.1285
EC129=41440.0305,-160425.1020
EC130=41440.0437,-256680.0755
EC131=41440.0570,-352935.0490
EC132=32275.1155,-417105.0000
EC133=32275.1043,-320850.0571
EC134=32275.0930,-224595.1142
EC135=32275.0818,-128340.1714
EC136=32275.0716,-32085.1142
EC137=32275.0614,64169.9429
EC138=32275.0512,160425.0000
EC139=32275.0624,256680.0490
EC140=32275.0737,352935.0979
EC141=32275.0849,449190.1469
EC142=32275.0951,545445.0979
EC143=32275.1053,641700.0490
EC144=32275.1155,737955.0000
EC145=32551.5987,673785.0490
EC146=32551.5844,577530.0898
EC147=32551.5701,481275.1306
EC148=32551.5558,385020.1714
EC149=32551.5487,288765.0959
EC150=32551.5416,192510.0204
EC151=32551.5344,96254.9449
EC152=32551.5487,-0.0938
EC153=32551.5630,-96255.1326
EC154=32551.5772,-192510.1714
EC155=32551.5844,-288765.0979
EC156=32551.5915,-385020.0245
EC157=32551.5987,-481274.9510
EC158=36650.1183,-545444.9021
EC159=36650.1152,-449189.9755
EC160=36650.1121,-352935.0490
EC161=36650.1091,-256680.1224
EC162=36650.0948,-160425.1132
EC163=36650.0805,-64170.1040
EC164=36650.0662,32084.9051
EC165=36650.0683,128339.9776
EC166=36650.0703,224595.0500
EC167=36650.0724,320850.1224
EC168=36650.0877,417105.1142
EC169=36650.1030,513360.1061
EC170=36650.1183,609615.0979
EC171=37831.4186,545445.0979
EC172=37831.4043,449190.0898
EC173=37831.3900,352935.0816
EC174=37831.3757,256680.0734
EC175=37831.3778,160425.0071
EC176=37831.3798,64169.9408
EC177=37831.3818,-32085.1255
EC178=37831.3982,-128340.1081
EC179=37831.4145,-224595.0908
EC180=37831.4308,-320850.0734
EC181=37831.4267,-417105.0163
EC182=37831.4226,-513359.9592
EC183=37831.4186,-609614.9021
EC184=10201.1591,-673784.5104
EC185=10201.1668,-577529.7144
EC186=10201.1744,-481274.9184
EC187=10201.1821,-385020.1224
EC188=10201.1693,-288765.2448
EC189=10201.1566,-192510.3672
EC190=10201.1438,-96255.4896
EC191=10201.1359,-0.2897
EC192=10201.1280,96254.9102
EC193=10201.1201,192510.1102
EC194=10201.1331,288765.2366
EC195=10201.1461,385020.3631
EC196=10201.1591,481275.4896
EC197=13912.1400,417105.3917
EC198=13912.1309,320850.2448
EC199=13912.1217,224595.0979
EC200=13912.1125,128339.9510
EC201=13912.1247,32084.8409
EC202=13912.1370,-64170.2693
EC203=13912.1492,-160425.3794
EC204=13912.1584,-256680.2366
EC205=13912.1676,-352935.0938
EC206=13912.1768,-449189.9510
EC207=13912.1645,-545444.8368
EC208=13912.1523,-641699.7226
EC209=13912.1400,-737954.6083
EC210=14885.1386,-802124.7063
EC211=14885.1533,-705869.7552
EC212=14885.1681,-609614.8042
EC213=14885.1829,-513359.8531
EC214=14885.1778,-417105.0082
EC215=14885.1727,-320850.1632
EC216=14885.1676,-224595.3182
EC217=14885.1533,-128340.2672
EC218=14885.1391,-32085.2162
EC219=14885.1248,64169.8348
EC220=14885.1294,160424.9959
EC221=14885.1340,256680.1571
EC222=14885.1386,352935.3182
EC223=18201.2846,288765.1958
EC224=18201.2846,192510.1306
EC225=18201.2846,96255.0653
EC226=18201.2846,0.0000
EC227=18201.3004,-96255.0653
EC228=18201.3162,-192510.1306
EC229=18201.3320,-288765.1958
EC230=18201.3310,-385020.1306
EC231=18201.3300,-481275.0653
EC232=18201.3289,-577530.0000
EC233=18201.3141,-673784.9347
EC234=18201.2994,-770039.8694
EC235=18201.2846,-866294.8042
EC236=7239.4892,-930464.7063
EC237=7239.5034,-834209.6083
EC238=7239.5177,-737954.5104
EC239=7239.5320,-641699.4125
EC240=7239.5374,-545444.6981
EC241=7239.5427,-449189.9837
EC242=7239.5481,-352935.2693
EC243=7239.5340,-256680.3835
EC244=7239.5200,-160425.4977
EC245=7239.5060,-64170.6120
EC246=7239.5004,32084.6818
EC247=7239.4948,128339.9755
EC248=7239.4892,224595.2693
EC249=-8224.9849,160424.9510
EC250=-8224.9747,64170.2611
EC251=-8224.9645,-32084.4288
EC252=-8224.9543,-128339.1188
EC253=-8224.9431,-224594.3962
EC254=-8224.9319,-320849.6736
EC255=-8224.9207,-417104.9510
EC256=-8224.9309,-513360.2611
EC257=-8224.9411,-609615.5712
EC258=-8224.9513,-705870.8812
EC259=-8224.9625,-802125.6201
EC260=-8224.9737,-898380.3590
EC261=-8224.9849,-994635.0979
EC262=-4750.0637,-1058804.4125
EC263=-4750.0566,-962550.2122
EC264=-4750.0494,-866296.0118
EC265=-4750.0423,-770041.8114
EC266=-4750.0290,-673786.3871
EC267=-4750.0158,-577530.9628
EC268=-4750.0025,-481275.5385
EC269=-4750.0097,-385019.7593
EC270=-4750.0168,-288763.9800
EC271=-4750.0239,-192508.2008
EC272=-4750.0372,-96253.6190
EC273=-4750.0505,0.9628
EC274=-4750.0637,96255.5447
EC275=-3533.4882,32645.5640
EC276=-3533.4727,-63998.4212
EC277=-3533.4573,-160642.4064
EC278=-3533.4419,-257286.3916
EC279=-3533.4403,-353524.8928
EC280=-3533.4388,-449763.3940
EC281=-3533.4373,-546001.8953
EC282=-3533.4517,-641870.3732
EC283=-3533.4661,-737738.8512
EC284=-3533.4805,-833607.3292
EC285=-3533.4831,-929876.3638
EC286=-3533.4856,-1026145.3983
EC287=-3533.4882,-1122414.4329
EC288=-3195.0077,-1186825.3054
EC289=-3195.0071,-1090424.1826
EC290=-3195.0066,-994023.0598
EC291=-3195.0060,-897621.9370
EC292=-3194.9949,-801725.3083
EC293=-3194.9838,-705828.6796
EC294=-3194.9727,-609932.0509
EC295=-3194.9659,-513824.9280
EC296=-3194.9591,-417717.8051
EC297=-3194.9523,-321610.6822
EC298=-3194.9707,-224995.5699
EC299=-3194.9892,-128380.4575
EC300=-3195.0077,-31765.3452
EC301=-20577.2782,-96254.7001
EC302=-20577.2654,-192509.7756
EC303=-20577.2527,-288764.8511
EC304=-20577.2399,-385019.9266
EC305=-20577.2481,-481275.0490
EC306=-20577.2563,-577530.1714
EC307=-20577.2644,-673785.2937
EC308=-20577.2772,-770040.2285
EC309=-20577.2899,-866295.1632
EC310=-20577.3027,-962550.0979
EC311=-20577.2945,-1058804.9674
EC312=-20577.2863,-1155059.8368
EC313=-20577.2782,-1251314.7063
EC314=-26008.5751,-1315484.8042
EC315=-26008.5863,-1219229.8694
EC316=-26008.5975,-1122974.9347
EC317=-26008.6088,-1026720.0000
EC318=-26008.5996,-930465.0816
EC319=-26008.5904,-834210.1632
EC320=-26008.5812,-737955.2448
EC321=-26008.5700,-641700.1795
EC322=-26008.5588,-545445.1142
EC323=-26008.5476,-449190.0490
EC324=-26008.5567,-352934.9551
EC325=-26008.5659,-256679.8613
EC326=-26008.5751,-160424.7675
EC327=-23105.8596,-224594.7552
EC328=-23105.8550,-320849.8858
EC329=-23105.8504,-417105.0163
EC330=-23105.8458,-513360.1469
EC331=-23105.8601,-609615.1795
EC332=-23105.8744,-705870.2122
EC333=-23105.8886,-802125.2448
EC334=-23105.8932,-898380.1306
EC335=-23105.8978,-994635.0163
EC336=-23105.9024,-1090889.9021
EC337=-23105.8881,-1187144.8694
EC338=-23105.8738,-1283399.8368
EC339=-23105.8596,-1379654.8042
EC340=-21969.0956,-1443824.8042
EC341=-21969.1109,-1347569.8694
EC342=-21969.1262,-1251314.9347
EC343=-21969.1415,-1155060.0000
EC344=-21969.1415,-1058805.0653
EC345=-21969.1415,-962550.1306
EC346=-21969.1415,-866295.1958
EC347=-21969.1267,-770040.1306
EC348=-21969.1119,-673785.0653
EC349=-21969.0971,-577530.0000
EC350=-21969.0966,-481274.9347
EC351=-21969.0961,-385019.8694
EC352=-21969.0956,-288764.8042
EC353=-26993.8483,-352934.9021
EC354=-26993.8544,-449190.0000
EC355=-26993.8605,-545445.0979
EC356=-26993.8666,-641700.1958
EC357=-26993.8799,-737955.1632
EC358=-26993.8931,-834210.1306
EC359=-26993.9064,-930465.0979
EC360=-26993.9013,-1026720.0000
EC361=-26993.8962,-1122974.9021
EC362=-26993.8911,-1219229.8042
EC363=-26993.8768,-1315484.8368
EC364=-26993.8625,-1411739.8694
EC365=-26993.8483,-1507994.9021
EC366=-45055.3781,-1572165.0000
EC367=-45055.3894,-1475909.9674
EC368=-45055.4006,-1379654.9347
EC369=-45055.4118,-1283399.9021
EC370=-45055.4210,-1187144.9347
EC371=-45055.4302,-1090889.9674
EC372=-45055.4393,-994635.0000
EC373=-45055.4291,-898380.0490
EC374=-45055.4189,-802125.0979
EC375=-45055.4087,-705870.1469
EC376=-45055.3985,-609615.0979
EC377=-45055.3883,-513360.0490
EC378=-45055.3781,-417105.0000
EC379=-45076.9226,-481275.0490
EC380=-45076.9349,-577530.0816
EC381=-45076.9471,-673785.1142
EC382=-45076.9594,-770040.1469
EC383=-45076.9665,-866295.0979
EC384=-45076.9736,-962550.0490
EC385=-45076.9808,-1058805.0000
EC386=-45076.9675,-1155059.9674
EC387=-45076.9543,-1251314.9347
EC388=-45076.9410,-1347569.9021
EC389=-45076.9349,-1443824.9347
EC390=-45076.9288,-1540079.9674
EC391=-45076.9226,-1636335.0000
EC392=-42057.8221,-1700505.0000
EC393=-42057.8252,-1604249.9674
EC394=-42057.8282,-1507994.9347
EC395=-42057.8313,-1411739.9021
EC396=-42057.8456,-1315484.9021
EC397=-42057.8598,-1219229.9021
EC398=-42057.8741,-1122974.9021
EC399=-42057.8721,-1026719.9674
EC400=-42057.8700,-930465.0326
EC401=-42057.8680,-834210.0979
EC402=-42057.8527,-737955.0979
EC403=-42057.8374,-641700.0979
EC404=-42057.8221,-545445.0979
EC405=-45068.6488,-609615.0979
EC406=-45068.6631,-705870.0979
EC407=-45068.6773,-802125.0979
EC408=-45068.6916,-898380.0979
EC409=-45068.6885,-994635.0326
EC410=-45068.6855,-1090889.9674
EC411=-45068.6824,-1187144.9021
EC412=-45068.6681,-1283399.9021
EC413=-45068.6539,-1379654.9021
EC414=-45068.6396,-1475909.9021
EC415=-45068.6427,-1572165.0000
EC416=-45068.6457,-1668420.0979
EC417=-45068.6488,-1764675.1958
EC418=-50107.1800,-1828845.1958
EC419=-50107.1719,-1732590.1306
EC420=-50107.1637,-1636335.0653
EC421=-50107.1555,-1540080.0000
EC422=-50107.1678,-1443824.9674
EC423=-50107.1800,-1347569.9347
EC424=-50107.1923,-1251314.9021
EC425=-50107.2004,-1155059.9347
EC426=-50107.2086,-1058804.9674
EC427=-50107.2167,-962550.0000
EC428=-50107.2045,-866295.0326
EC429=-50107.1923,-770040.0653
EC430=-50107.1800,-673785.0979
EC431=-64538.6585,-737955.0979
EC432=-64538.6667,-834210.0653
EC433=-64538.6749,-930465.0326
EC434=-64538.6830,-1026720.0000
EC435=-64538.6708,-1122974.9674
EC436=-64538.6585,-1219229.9347
EC437=-64538.6463,-1315484.9021
EC438=-64538.6381,-1411739.9347
EC439=-64538.6300,-1507994.9674
EC440=-64538.6218,-1604250.0000
EC441=-64538.6341,-1700505.0000
EC442=-64538.6463,-1796760.0000
EC443=-64538.6585,-1893015.0000
EC444=-65800.7790,-1957185.0000
EC445=-65800.7647,-1860930.0000
EC446=-65800.7505,-1764675.0000
EC447=-65800.7362,-1668420.0000
EC448=-65800.7403,-1572164.9674
EC449=-65800.7443,-1475909.9347
EC450=-65800.7484,-1379654.9021
EC451=-65800.7627,-1283399.9347
EC452=-65800.7770,-1187144.9674
EC453=-65800.7913,-1090890.0000
EC454=-65800.7872,-994635.0326
EC455=-65800.7831,-898380.0653
EC456=-65800.7790,-802125.0979
EC457=-67920.0286,-866295.0979
EC458=-67920.0286,-962550.0653
EC459=-67920.0286,-1058805.0326
EC460=-67920.0286,-1155060.0000
EC461=-67920.0123,-1251314.9674
EC462=-67919.9960,-1347569.9347
EC463=-67919.9797,-1443824.9021
EC464=-67919.9817,-1540079.9347
EC465=-67919.9837,-1636334.9674
EC466=-67919.9858,-1732590.0000
EC467=-67920.0001,-1828845.0000
EC468=-67920.0143,-1925100.0000
EC469=-67920.0286,-2021355.0000
EC470=-70223.0414,-2085525.0000
EC471=-70223.0271,-1989270.0000
EC472=-70223.0129,-1893015.0000
EC473=-70222.9986,-1796760.0000
EC474=-70222.9925,-1700505.0000
EC475=-70222.9863,-1604250.0000
EC476=-70222.9802,-1507995.0000
EC477=-70222.9945,-1411739.9674
EC478=-70223.0088,-1315484.9347
EC479=-70223.0231,-1219229.9021
EC480=-70223.0292,-1122974.9347
EC481=-70223.0353,-1026719.9674
EC482=-70223.0414,-930465.0000
EC483=-74613.5241,-994635.0000
EC484=-74613.5139,-1090889.9674
EC485=-74613.5037,-1187144.9347
EC486=-74613.4935,-1283399.9021
EC487=-74613.4833,-1379654.9347
EC488=-74613.4731,-1475909.9674
EC489=-74613.4629,-1572165.0000
EC490=-74613.4731,-1668420.0000
EC491=-74613.4833,-1764675.0000
EC492=-74613.4935,-1860930.0000
EC493=-74613.5037,-1957185.0000
EC494=-74613.5139,-2053440.0000
EC495=-74613.5241,-2149695.0000
EC496=-73913.5190,-2213865.0000
EC497=-73913.5128,-2117610.0000
EC498=-73913.5067,-2021355.0000
EC499=-73913.5006,-1925100.0000
EC500=-73913.4884,-1828845.0000
EC501=-73913.4761,-1732590.0000
EC502=-73913.4639,-1636335.0000
EC503=-73913.4700,-1540079.9674
EC504=-73913.4761,-1443824.9347
EC505=-73913.4822,-1347569.9021
EC506=-73913.4945,-1251314.9347
EC507=-73913.5067,-1155059.9674
EC508=-73913.5190,-1058805.0000
EC509=-84539.5945,-1122975.0000
EC510=-84539.5802,-1219229.9674
EC511=-84539.5659,-1315484.9347
EC512=-84539.5517,-1411739.9021
EC513=-84539.5496,-1507994.9347
EC514=-84539.5476,-1604249.9674
EC515=-84539.5455,-1700505.0000
EC516=-84539.5578,-1796760.0000
EC517=-84539.5700,-1893015.0000
EC518=-84539.5823,-1989270.0000
EC519=-84539.5863,-2085525.0000
EC520=-84539.5904,-2181780.0000
EC521=-84539.5945,-2278035.0000
EC522=-74484.6548,-2342205.0000
EC523=-74484.6589,-2245950.0000
EC524=-74484.6630,-2149695.0000
EC525=-74484.6671,-2053440.0000
EC526=-74484.6507,-1957185.0000
EC527=-74484.6344,-1860930.0000
EC528=-74484.6181,-1764675.0000
EC529=-74484.6161,-1668420.0000
EC530=-74484.6140,-1572165.0000
EC531=-74484.6120,-1475910.0000
EC532=-74484.6263,-1379654.9674
EC533=-74484.6405,-1283399.9347
EC534=-74484.6548,-1187144.9021
EC535=-48864.6671,-1251314.9021
EC536=-48864.6539,-1347569.9347
EC537=-48864.6406,-1443824.9674
EC538=-48864.6274,-1540080.0000
EC539=-48864.6365,-1636335.0653
EC540=-48864.6457,-1732590.1306
EC541=-48864.6549,-1828845.1958
EC542=-48864.6671,-1925100.1306
EC543=-48864.6794,-2021355.0653
EC544=-48864.6916,-2117610.0000
EC545=-48864.6835,-2213864.9347
EC546=-48864.6753,-2310119.8694
EC547=-48864.6671,-2406374.8042
EC548=-23588.2655,-2470544.8042
EC549=-23588.2772,-2374289.8694
EC550=-23588.2889,-2278034.9347
EC551=-23588.3007,-2181780.0000
EC552=-23588.2910,-2085525.0653
EC553=-23588.2813,-1989270.1306
EC554=-23588.2716,-1893015.1958
EC555=-23588.2604,-1796760.1306
EC556=-23588.2492,-1700505.0653
EC557=-23588.2379,-1604250.0000
EC558=-23588.2471,-1507994.9021
EC559=-23588.2563,-1411739.8042
EC560=-23588.2655,-1315484.7063
EC561=-3927.8040,-1380243.7668
EC562=-3927.7966,-1476558.6585
EC563=-3927.7893,-1572873.5503
EC564=-3927.7819,-1669188.4420
EC565=-3927.7989,-1764992.7036
EC566=-3927.8160,-1860796.9653
EC567=-3927.8331,-1956601.2269
EC568=-3927.8349,-2052793.0387
EC569=-3927.8367,-2148984.8504
EC570=-3927.8385,-2245176.6622
EC571=-3927.8270,-2341885.7297
EC572=-3927.8155,-2438594.7972
EC573=-3927.8040,-2535303.8647
EC574=-1941.3856,-2599702.0082
EC575=-1941.4014,-2502999.2726
EC576=-1941.4171,-2406296.5369
EC577=-1941.4329,-2309593.8013
EC578=-1941.4327,-2213243.4315
EC579=-1941.4325,-2116893.0616
EC580=-1941.4323,-2020542.6918
EC581=-1941.4179,-1924732.2941
EC582=-1941.4035,-1828921.8964
EC583=-1941.3891,-1733111.4987
EC584=-1941.3879,-1636955.0019
EC585=-1941.3868,-1540798.5050
EC586=-1941.3856,-1444642.0082
EC587=-1711.1944,-1508940.7673
EC588=-1711.2003,-1604951.3372
EC589=-1711.2063,-1700961.9071
EC590=-1711.2123,-1796972.4770
EC591=-1711.2260,-1892842.1462
EC592=-1711.2396,-1988711.8155
EC593=-1711.2533,-2084581.4848
EC594=-1711.2480,-2181079.3809
EC595=-1711.2428,-2277577.2770
EC596=-1711.2376,-2374075.1731
EC597=-1711.2232,-2470717.0704
EC598=-1711.2088,-2567358.9678
EC599=-1711.1944,-2664000.8652
EC600=-1484.9182,-2728185.1609
EC601=-1484.9288,-2631651.1013
EC602=-1484.9395,-2535117.0417
EC603=-1484.9501,-2438582.9821
EC604=-1484.9608,-2341966.5428
EC605=-1484.9715,-2245350.1035
EC606=-1484.9822,-2148733.6642
EC607=-1484.9703,-2052758.5724
EC608=-1484.9585,-1956783.4806
EC609=-1484.9466,-1860808.3888
EC610=-1484.9371,-1764913.9795
EC611=-1484.9276,-1669019.5702
EC612=-1484.9182,-1573125.1609
EC613=-1257.8348,-1637193.8182
EC614=-1257.8471,-1733015.4109
EC615=-1257.8594,-1828837.0036
EC616=-1257.8717,-1924658.5963
EC617=-1257.8798,-2020773.0547
EC618=-1257.8880,-2116887.5131
EC619=-1257.8961,-2213001.9715
EC620=-1257.8818,-2309693.2183
EC621=-1257.8675,-2406384.4652
EC622=-1257.8531,-2503075.7120
EC623=-1257.8470,-2599468.4467
EC624=-1257.8409,-2695861.1814
EC625=-1257.8348,-2792253.9161
EC626=-1145.6476,-2856219.6640
EC627=-1145.6499,-2759984.3777
EC628=-1145.6522,-2663749.0914
EC629=-1145.6545,-2567513.8051
EC630=-1145.6693,-2470800.9515
EC631=-1145.6841,-2374088.0979
EC632=-1145.6990,-2277375.2444
EC633=-1145.6969,-2181103.9251
EC634=-1145.6949,-2084832.6058
EC635=-1145.6928,-1988561.2865
EC636=-1145.6778,-1892760.7457
EC637=-1145.6627,-1796960.2049
EC638=-1145.6476,-1701159.6640
//INST
///DATE 0000/00/00 00:00
///ATTR SC,RW,RJ
////FRAME USER 4
///GROUP1 RB1
///GROUP2 ST1
///COMM ADA_SLICER
NOP
SKILLSND ATTR=3 "corrpath"
MOVJ P0  VJ=10.0  +MOVJ EC0 VJ=10.0
'LAYER_1
SMOVL C0 V=30.0  +MOVJ EC1
MACRO1 MJ#(16)
MACRO1 MJ#(9) ARGF30 ARGF0
WVON AMP=3.1 FREQ=2.5 ANGL=0.0 DIR=0
SMOVL C1 V=10.0  +MOVJ EC2
SMOVL C2 V=10.0  +MOVJ EC3
SMOVL C3 V=10.0  +MOVJ EC4
SMOVL C4 V=10.0  +MOVJ EC5
SMOVL C5 V=10.0  +MOVJ EC6
SMOVL C6 V=10.0  +MOVJ EC7
SMOVL C7 V=10.0  +MOVJ EC8
SMOVL C8 V=10.0  +MOVJ EC9
SMOVL C9 V=10.0  +MOVJ EC10
SMOVL C10 V=10.0  +MOVJ EC11
SMOVL C11 V=10.0  +MOVJ EC12
SMOVL C12 V=10.0  +MOVJ EC13
WVOF
MACRO1 MJ#(10)
SMOVL C13 V=30.0  +MOVJ EC14
'LAYER_2
SMOVL C14 V=30.0  +MOVJ EC15
MACRO1 MJ#(16)
MACRO1 MJ#(9) ARGF30 ARGF0
WVON AMP=3.1 FREQ=2.5 ANGL=0.0 DIR=0
SMOVL C15 V=10.0  +MOVJ EC16
SMOVL C16 V=10.0  +MOVJ EC17
SMOVL C17 V=10.0  +MOVJ EC18
SMOVL C18 V=10.0  +MOVJ EC19
SMOVL C19 V=10.0  +MOVJ EC20
SMOVL C20 V=10.0  +MOVJ EC21
SMOVL C21 V=10.0  +MOVJ EC22
SMOVL C22 V=10.0  +MOVJ EC23
SMOVL C23 V=10.0  +MOVJ EC24
SMOVL C24 V=10.0  +MOVJ EC25
SMOVL C25 V=10.0  +MOVJ EC26
SMOVL C26 V=10.0  +MOVJ EC27
WVOF
MACRO1 MJ#(10)
'LAYER_3
SMOVL C27 V=30.0  +MOVJ EC28
MACRO1 MJ#(16)
MACRO1 MJ#(9) ARGF30 ARGF0
WVON AMP=3.1 FREQ=2.5 ANGL=0.0 DIR=0
SMOVL C28 V=10.0  +MOVJ EC29
SMOVL C29 V=10.0  +MOVJ EC30
SMOVL C30 V=10.0  +MOVJ EC31
SMOVL C31 V=10.0  +MOVJ EC32
SMOVL C32 V=10.0  +MOVJ EC33
SMOVL C33 V=10.0  +MOVJ EC34
SMOVL C34 V=10.0  +MOVJ EC35
SMOVL C35 V=10.0  +MOVJ EC36
SMOVL C36 V=10.0  +MOVJ EC37
SMOVL C37 V=10.0  +MOVJ EC38
SMOVL C38 V=10.0  +MOVJ EC39
SMOVL C39 V=10.0  +MOVJ EC40
WVOF
MACRO1 MJ#(10)
'LAYER_4
SMOVL C40 V=30.0  +MOVJ EC41
MACRO1 MJ#(16)
MACRO1 MJ#(9) ARGF30 ARGF0
WVON AMP=3.1 FREQ=2.5 ANGL=0.0 DIR=0
SMOVL C41 V=10.0  +MOVJ EC42
SMOVL C42 V=10.0  +MOVJ EC43
SMOVL C43 V=10.0  +MOVJ EC44
SMOVL C44 V=10.0  +MOVJ EC45
SMOVL C45 V=10.0  +MOVJ EC46
SMOVL C46 V=10.0  +MOVJ EC47
SMOVL C47 V=10.0  +MOVJ EC48
SMOVL C48 V=10.0  +MOVJ EC49
SMOVL C49 V=10.0  +MOVJ EC50
SMOVL C50 V=10.0  +MOVJ EC51
SMOVL C51 V=10.0  +MOVJ EC52
SMOVL C52 V=10.0  +MOVJ EC53
WVOF
MACRO1 MJ#(10)
'LAYER_5
SMOVL C53 V=30.0  +MOVJ EC54
MACRO1 MJ#(16)
MACRO1 MJ#(9) ARGF30 ARGF0
WVON AMP=3.1 FREQ=2.5 ANGL=0.0 DIR=0
SMOVL C54 V=10.0  +MOVJ EC55
SMOVL C55 V=10.0  +MOVJ EC56
SMOVL C56 V=10.0  +MOVJ EC57
SMOVL C57 V=10.0  +MOVJ EC58
SMOVL C58 V=10.0  +MOVJ EC59
SMOVL C59 V=10.0  +MOVJ EC60
SMOVL C60 V=10.0  +MOVJ EC61
SMOVL C61 V=10.0  +MOVJ EC62
SMOVL C62 V=10.0  +MOVJ EC63
SMOVL C63 V=10.0  +MOVJ EC64
SMOVL C64 V=10.0  +MOVJ EC65
SMOVL C65 V=10.0  +MOVJ EC66
WVOF
MACRO1 MJ#(10)
'LAYER_6
SMOVL C66 V=30.0  +MOVJ EC67
MACRO1 MJ#(16)
MACRO1 MJ#(9) ARGF30 ARGF0
WVON AMP=3.1 FREQ=2.5 ANGL=0.0 DIR=0
SMOVL C67 V=10.0  +MOVJ EC68
SMOVL C68 V=10.0  +MOVJ EC69
SMOVL C69 V=10.0  +MOVJ EC70
SMOVL C70 V=10.0  +MOVJ EC71
SMOVL C71 V=10.0  +MOVJ EC72
SMOVL C72 V=10.0  +MOVJ EC73
SMOVL C73 V=10.0  +MOVJ EC74
SMOVL C74 V=10.0  +MOVJ EC75
SMOVL C75 V=10.0  +MOVJ EC76
SMOVL C76 V=10.0  +MOVJ EC77
SMOVL C77 V=10.0  +MOVJ EC78
SMOVL C78 V=10.0  +MOVJ EC79
WVOF
MACRO1 MJ#(10)
'LAYER_7
SMOVL C79 V=30.0  +MOVJ EC80
MACRO1 MJ#(16)
MACRO1 MJ#(9) ARGF30 ARGF0
WVON AMP=3.1 FREQ=2.5 ANGL=0.0 DIR=0
SMOVL C80 V=10.0  +MOVJ EC81
SMOVL C81 V=10.0  +MOVJ EC82
SMOVL C82 V=10.0  +MOVJ EC83
SMOVL C83 V=10.0  +MOVJ EC84
SMOVL C84 V=10.0  +MOVJ EC85
SMOVL C85 V=10.0  +MOVJ EC86
SMOVL C86 V=10.0  +MOVJ EC87
SMOVL C87 V=10.0  +MOVJ EC88
SMOVL C88 V=10.0  +MOVJ EC89
SMOVL C89 V=10.0  +MOVJ EC90
SMOVL C90 V=10.0  +MOVJ EC91
SMOVL C91 V=10.0  +MOVJ EC92
WVOF
MACRO1 MJ#(10)
'LAYER_8
SMOVL C92 V=30.0  +MOVJ EC93
MACRO1 MJ#(16)
MACRO1 MJ#(9) ARGF30 ARGF0
WVON AMP=3.1 FREQ=2.5 ANGL=0.0 DIR=0
SMOVL C93 V=10.0  +MOVJ EC94
SMOVL C94 V=10.0  +MOVJ EC95
SMOVL C95 V=10.0  +MOVJ EC96
SMOVL C96 V=10.0  +MOVJ EC97
SMOVL C97 V=10.0  +MOVJ EC98
SMOVL C98 V=10.0  +MOVJ EC99
SMOVL C99 V=10.0  +MOVJ EC100
SMOVL C100 V=10.0  +MOVJ EC101
SMOVL C101 V=10.0  +MOVJ EC102
SMOVL C102 V=10.0  +MOVJ EC103
SMOVL C103 V=10.0  +MOVJ EC104
SMOVL C104 V=10.0  +MOVJ EC105
WVOF
MACRO1 MJ#(10)
'LAYER_9
SMOVL C105 V=30.0  +MOVJ EC106
MACRO1 MJ#(16)
MACRO1 MJ#(9) ARGF30 ARGF0
WVON AMP=3.1 FREQ=2.5 ANGL=0.0 DIR=0
SMOVL C106 V=10.0  +MOVJ EC107
SMOVL C107 V=10.0  +MOVJ EC108
SMOVL C108 V=10.0  +MOVJ EC109
SMOVL C109 V=10.0  +MOVJ EC110
SMOVL C110 V=10.0  +MOVJ EC111
SMOVL C111 V=10.0  +MOVJ EC112
SMOVL C112 V=10.0  +MOVJ EC113
SMOVL C113 V=10.0  +MOVJ EC114
SMOVL C114 V=10.0  +MOVJ EC115
SMOVL C115 V=10.0  +MOVJ EC116
SMOVL C116 V=10.0  +MOVJ EC117
SMOVL C117 V=10.0  +MOVJ EC118
WVOF
MACRO1 MJ#(10)
'LAYER_10
SMOVL C118 V=30.0  +MOVJ EC119
MACRO1 MJ#(16)
MACRO1 MJ#(9) ARGF30 ARGF0
WVON AMP=3.1 FREQ=2.5 ANGL=0.0 DIR=0
SMOVL C119 V=10.0  +MOVJ EC120
SMOVL C120 V=10.0  +MOVJ EC121
SMOVL C121 V=10.0  +MOVJ EC122
SMOVL C122 V=10.0  +MOVJ EC123
SMOVL C123 V=10.0  +MOVJ EC124
SMOVL C124 V=10.0  +MOVJ EC125
SMOVL C125 V=10.0  +MOVJ EC126
SMOVL C126 V=10.0  +MOVJ EC127
SMOVL C127 V=10.0  +MOVJ EC128
SMOVL C128 V=10.0  +MOVJ EC129
SMOVL C129 V=10.0  +MOVJ EC130
SMOVL C130 V=10.0  +MOVJ EC131
WVOF
MACRO1 MJ#(10)
'LAYER_11
SMOVL C131 V=30.0  +MOVJ EC132
MACRO1 MJ#(16)
MACRO1 MJ#(9) ARGF30 ARGF0
WVON AMP=3.1 FREQ=2.5 ANGL=0.0 DIR=0
SMOVL C132 V=10.0  +MOVJ EC133
SMOVL C133 V=10.0  +MOVJ EC134
SMOVL C134 V=10.0  +MOVJ EC135
SMOVL C135 V=10.0  +MOVJ EC136
SMOVL C136 V=10.0  +MOVJ EC137
SMOVL C137 V=10.0  +MOVJ EC138
SMOVL C138 V=10.0  +MOVJ EC139
SMOVL C139 V=10.0  +MOVJ EC140
SMOVL C140 V=10.0  +MOVJ EC141
SMOVL C141 V=10.0  +MOVJ EC142
SMOVL C142 V=10.0  +MOVJ EC143
SMOVL C143 V=10.0  +MOVJ EC144
WVOF
MACRO1 MJ#(10)
'LAYER_12
SMOVL C144 V=30.0  +MOVJ EC145
MACRO1 MJ#(16)
MACRO1 MJ#(9) ARGF30 ARGF0
WVON AMP=3.1 FREQ=2.5 ANGL=0.0 DIR=0
SMOVL C145 V=10.0  +MOVJ EC146
SMOVL C146 V=10.0  +MOVJ EC147
SMOVL C147 V=10.0  +MOVJ EC148
SMOVL C148 V=10.0  +MOVJ EC149
SMOVL C149 V=10.0  +MOVJ EC150
SMOVL C150 V=10.0  +MOVJ EC151
SMOVL C151 V=10.0  +MOVJ EC152
SMOVL C152 V=10.0  +MOVJ EC153
SMOVL C153 V=10.0  +MOVJ EC154
SMOVL C154 V=10.0  +MOVJ EC155
SMOVL C155 V=10.0  +MOVJ EC156
SMOVL C156 V=10.0  +MOVJ EC157
WVOF
MACRO1 MJ#(10)
'LAYER_13
SMOVL C157 V=30.0  +MOVJ EC158
MACRO1 MJ#(16)
MACRO1 MJ#(9) ARGF30 ARGF0
WVON AMP=3.1 FREQ=2.5 ANGL=0.0 DIR=0
SMOVL C158 V=10.0  +MOVJ EC159
SMOVL C159 V=10.0  +MOVJ EC160
SMOVL C160 V=10.0  +MOVJ EC161
SMOVL C161 V=10.0  +MOVJ EC162
SMOVL C162 V=10.0  +MOVJ EC163
SMOVL C163 V=10.0  +MOVJ EC164
SMOVL C164 V=10.0  +MOVJ EC165
SMOVL C165 V=10.0  +MOVJ EC166
SMOVL C166 V=10.0  +MOVJ EC167
SMOVL C167 V=10.0  +MOVJ EC168
SMOVL C168 V=10.0  +MOVJ EC169
SMOVL C169 V=10.0  +MOVJ EC170
WVOF
MACRO1 MJ#(10)
'LAYER_14
SMOVL C170 V=30.0  +MOVJ EC171
MACRO1 MJ#(16)
MACRO1 MJ#(9) ARGF30 ARGF0
WVON AMP=3.1 FREQ=2.5 ANGL=0.0 DIR=0
SMOVL C171 V=10.0  +MOVJ EC172
SMOVL C172 V=10.0  +MOVJ EC173
SMOVL C173 V=10.0  +MOVJ EC174
SMOVL C174 V=10.0  +MOVJ EC175
SMOVL C175 V=10.0  +MOVJ EC176
SMOVL C176 V=10.0  +MOVJ EC177
SMOVL C177 V=10.0  +MOVJ EC178
SMOVL C178 V=10.0  +MOVJ EC179
SMOVL C179 V=10.0  +MOVJ EC180
SMOVL C180 V=10.0  +MOVJ EC181
SMOVL C181 V=10.0  +MOVJ EC182
SMOVL C182 V=10.0  +MOVJ EC183
WVOF
MACRO1 MJ#(10)
'LAYER_15
SMOVL C183 V=30.0  +MOVJ EC184
MACRO1 MJ#(16)
MACRO1 MJ#(9) ARGF30 ARGF0
WVON AMP=3.1 FREQ=2.5 ANGL=0.0 DIR=0
SMOVL C184 V=10.0  +MOVJ EC185
SMOVL C185 V=10.0  +MOVJ EC186
SMOVL C186 V=10.0  +MOVJ EC187
SMOVL C187 V=10.0  +MOVJ EC188
SMOVL C188 V=10.0  +MOVJ EC189
SMOVL C189 V=10.0  +MOVJ EC190
SMOVL C190 V=10.0  +MOVJ EC191
SMOVL C191 V=10.0  +MOVJ EC192
SMOVL C192 V=10.0  +MOVJ EC193
SMOVL C193 V=10.0  +MOVJ EC194
SMOVL C194 V=10.0  +MOVJ EC195
SMOVL C195 V=10.0  +MOVJ EC196
WVOF
MACRO1 MJ#(10)
'LAYER_16
SMOVL C196 V=30.0  +MOVJ EC197
MACRO1 MJ#(16)
MACRO1 MJ#(9) ARGF30 ARGF0
WVON AMP=3.1 FREQ=2.5 ANGL=0.0 DIR=0
SMOVL C197 V=10.0  +MOVJ EC198
SMOVL C198 V=10.0  +MOVJ EC199
SMOVL C199 V=10.0  +MOVJ EC200
SMOVL C200 V=10.0  +MOVJ EC201
SMOVL C201 V=10.0  +MOVJ EC202
SMOVL C202 V=10.0  +MOVJ EC203
SMOVL C203 V=10.0  +MOVJ EC204
SMOVL C204 V=10.0  +MOVJ EC205
SMOVL C205 V=10.0  +MOVJ EC206
SMOVL C206 V=10.0  +MOVJ EC207
SMOVL C207 V=10.0  +MOVJ EC208
SMOVL C208 V=10.0  +MOVJ EC209
WVOF
MACRO1 MJ#(10)
'LAYER_17
SMOVL C209 V=30.0  +MOVJ EC210
MACRO1 MJ#(16)
MACRO1 MJ#(9) ARGF30 ARGF0
WVON AMP=3.1 FREQ=2.5 ANGL=0.0 DIR=0
SMOVL C210 V=10.0  +MOVJ EC211
SMOVL C211 V=10.0  +MOVJ EC212
SMOVL C212 V=10.0  +MOVJ EC213
SMOVL C213 V=10.0  +MOVJ EC214
SMOVL C214 V=10.0  +MOVJ EC215
SMOVL C215 V=10.0  +MOVJ EC216
SMOVL C216 V=10.0  +MOVJ EC217
SMOVL C217 V=10.0  +MOVJ EC218
SMOVL C218 V=10.0  +MOVJ EC219
SMOVL C219 V=10.0  +MOVJ EC220
SMOVL C220 V=10.0  +MOVJ EC221
SMOVL C221 V=10.0  +MOVJ EC222
WVOF
MACRO1 MJ#(10)
'LAYER_18
SMOVL C222 V=30.0  +MOVJ EC223
MACRO1 MJ#(16)
MACRO1 MJ#(9) ARGF30 ARGF0
WVON AMP=3.1 FREQ=2.5 ANGL=0.0 DIR=0
SMOVL C223 V=10.0  +MOVJ EC224
SMOVL C224 V=10.0  +MOVJ EC225
SMOVL C225 V=10.0  +MOVJ EC226
SMOVL C226 V=10.0  +MOVJ EC227
SMOVL C227 V=10.0  +MOVJ EC228
SMOVL C228 V=10.0  +MOVJ EC229
SMOVL C229 V=10.0  +MOVJ EC230
SMOVL C230 V=10.0  +MOVJ EC231
SMOVL C231 V=10.0  +MOVJ EC232
SMOVL C232 V=10.0  +MOVJ EC233
SMOVL C233 V=10.0  +MOVJ EC234
SMOVL C234 V=10.0  +MOVJ EC235
WVOF
MACRO1 MJ#(10)
'LAYER_19
SMOVL C235 V=30.0  +MOVJ EC236
MACRO1 MJ#(16)
MACRO1 MJ#(9) ARGF30 ARGF0
WVON AMP=3.1 FREQ=2.5 ANGL=0.0 DIR=0
SMOVL C236 V=10.0  +MOVJ EC237
SMOVL C237 V=10.0  +MOVJ EC238
SMOVL C238 V=10.0  +MOVJ EC239
SMOVL C239 V=10.0  +MOVJ EC240
SMOVL C240 V=10.0  +MOVJ EC241
SMOVL C241 V=10.0  +MOVJ EC242
SMOVL C242 V=10.0  +MOVJ EC243
SMOVL C243 V=10.0  +MOVJ EC244
SMOVL C244 V=10.0  +MOVJ EC245
SMOVL C245 V=10.0  +MOVJ EC246
SMOVL C246 V=10.0  +MOVJ EC247
SMOVL C247 V=10.0  +MOVJ EC248
WVOF
MACRO1 MJ#(10)
'LAYER_20
SMOVL C248 V=30.0  +MOVJ EC249
MACRO1 MJ#(16)
MACRO1 MJ#(9) ARGF30 ARGF0
WVON AMP=3.1 FREQ=2.5 ANGL=0.0 DIR=0
SMOVL C249 V=10.0  +MOVJ EC250
SMOVL C250 V=10.0  +MOVJ EC251
SMOVL C251 V=10.0  +MOVJ EC252
SMOVL C252 V=10.0  +MOVJ EC253
SMOVL C253 V=10.0  +MOVJ EC254
SMOVL C254 V=10.0  +MOVJ EC255
SMOVL C255 V=10.0  +MOVJ EC256
SMOVL C256 V=10.0  +MOVJ EC257
SMOVL C257 V=10.0  +MOVJ EC258
SMOVL C258 V=10.0  +MOVJ EC259
SMOVL C259 V=10.0  +MOVJ EC260
SMOVL C260 V=10.0  +MOVJ EC261
WVOF
MACRO1 MJ#(10)
'LAYER_21
SMOVL C261 V=30.0  +MOVJ EC262
MACRO1 MJ#(16)
MACRO1 MJ#(9) ARGF30 ARGF0
WVON AMP=3.1 FREQ=2.5 ANGL=0.0 DIR=0
SMOVL C262 V=10.0  +MOVJ EC263
SMOVL C263 V=10.0  +MOVJ EC264
SMOVL C264 V=10.0  +MOVJ EC265
SMOVL C265 V=10.0  +MOVJ EC266
SMOVL C266 V=10.0  +MOVJ EC267
SMOVL C267 V=10.0  +MOVJ EC268
SMOVL C268 V=10.0  +MOVJ EC269
SMOVL C269 V=10.0  +MOVJ EC270
SMOVL C270 V=10.0  +MOVJ EC271
SMOVL C271 V=10.0  +MOVJ EC272
SMOVL C272 V=10.0  +MOVJ EC273
SMOVL C273 V=10.0  +MOVJ EC274
WVOF
MACRO1 MJ#(10)
'LAYER_22
SMOVL C274 V=30.0  +MOVJ EC275
MACRO1 MJ#(16)
MACRO1 MJ#(9) ARGF30 ARGF0
WVON AMP=3.1 FREQ=2.5 ANGL=0.0 DIR=0
SMOVL C275 V=10.0  +MOVJ EC276
SMOVL C276 V=10.0  +MOVJ EC277
SMOVL C277 V=10.0  +MOVJ EC278
SMOVL C278 V=10.0  +MOVJ EC279
SMOVL C279 V=10.0  +MOVJ EC280
SMOVL C280 V=10.0  +MOVJ EC281
SMOVL C281 V=10.0  +MOVJ EC282
SMOVL C282 V=10.0  +MOVJ EC283
SMOVL C283 V=10.0  +MOVJ EC284
SMOVL C284 V=10.0  +MOVJ EC285
SMOVL C285 V=10.0  +MOVJ EC286
SMOVL C286 V=10.0  +MOVJ EC287
WVOF
MACRO1 MJ#(10)
'LAYER_23
SMOVL C287 V=30.0  +MOVJ EC288
MACRO1 MJ#(16)
MACRO1 MJ#(9) ARGF30 ARGF0
WVON AMP=3.1 FREQ=2.5 ANGL=0.0 DIR=0
SMOVL C288 V=10.0  +MOVJ EC289
SMOVL C289 V=10.0  +MOVJ EC290
SMOVL C290 V=10.0  +MOVJ EC291
SMOVL C291 V=10.0  +MOVJ EC292
SMOVL C292 V=10.0  +MOVJ EC293
SMOVL C293 V=10.0  +MOVJ EC294
SMOVL C294 V=10.0  +MOVJ EC295
SMOVL C295 V=10.0  +MOVJ EC296
SMOVL C296 V=10.0  +MOVJ EC297
SMOVL C297 V=10.0  +MOVJ EC298
SMOVL C298 V=10.0  +MOVJ EC299
SMOVL C299 V=10.0  +MOVJ EC300
WVOF
MACRO1 MJ#(10)
'LAYER_24
SMOVL C300 V=30.0  +MOVJ EC301
MACRO1 MJ#(16)
MACRO1 MJ#(9) ARGF30 ARGF0
WVON AMP=3.1 FREQ=2.5 ANGL=0.0 DIR=0
SMOVL C301 V=10.0  +MOVJ EC302
SMOVL C302 V=10.0  +MOVJ EC303
SMOVL C303 V=10.0  +MOVJ EC304
SMOVL C304 V=10.0  +MOVJ EC305
SMOVL C305 V=10.0  +MOVJ EC306
SMOVL C306 V=10.0  +MOVJ EC307
SMOVL C307 V=10.0  +MOVJ EC308
SMOVL C308 V=10.0  +MOVJ EC309
SMOVL C309 V=10.0  +MOVJ EC310
SMOVL C310 V=10.0  +MOVJ EC311
SMOVL C311 V=10.0  +MOVJ EC312
SMOVL C312 V=10.0  +MOVJ EC313
WVOF
MACRO1 MJ#(10)
'LAYER_25
SMOVL C313 V=30.0  +MOVJ EC314
MACRO1 MJ#(16)
MACRO1 MJ#(9) ARGF30 ARGF0
WVON AMP=3.1 FREQ=2.5 ANGL=0.0 DIR=0
SMOVL C314 V=10.0  +MOVJ EC315
SMOVL C315 V=10.0  +MOVJ EC316
SMOVL C316 V=10.0  +MOVJ EC317
SMOVL C317 V=10.0  +MOVJ EC318
SMOVL C318 V=10.0  +MOVJ EC319
SMOVL C319 V=10.0  +MOVJ EC320
SMOVL C320 V=10.0  +MOVJ EC321
SMOVL C321 V=10.0  +MOVJ EC322
SMOVL C322 V=10.0  +MOVJ EC323
SMOVL C323 V=10.0  +MOVJ EC324
SMOVL C324 V=10.0  +MOVJ EC325
SMOVL C325 V=10.0  +MOVJ EC326
WVOF
MACRO1 MJ#(10)
'LAYER_26
SMOVL C326 V=30.0  +MOVJ EC327
MACRO1 MJ#(16)
MACRO1 MJ#(9) ARGF30 ARGF0
WVON AMP=3.1 FREQ=2.5 ANGL=0.0 DIR=0
SMOVL C327 V=10.0  +MOVJ EC328
SMOVL C328 V=10.0  +MOVJ EC329
SMOVL C329 V=10.0  +MOVJ EC330
SMOVL C330 V=10.0  +MOVJ EC331
SMOVL C331 V=10.0  +MOVJ EC332
SMOVL C332 V=10.0  +MOVJ EC333
SMOVL C333 V=10.0  +MOVJ EC334
SMOVL C334 V=10.0  +MOVJ EC335
SMOVL C335 V=10.0  +MOVJ EC336
SMOVL C336 V=10.0  +MOVJ EC337
SMOVL C337 V=10.0  +MOVJ EC338
SMOVL C338 V=10.0  +MOVJ EC339
WVOF
MACRO1 MJ#(10)
'LAYER_27
SMOVL C339 V=30.0  +MOVJ EC340
MACRO1 MJ#(16)
MACRO1 MJ#(9) ARGF30 ARGF0
WVON AMP=3.1 FREQ=2.5 ANGL=0.0 DIR=0
SMOVL C340 V=10.0  +MOVJ EC341
SMOVL C341 V=10.0  +MOVJ EC342
SMOVL C342 V=10.0  +MOVJ EC343
SMOVL C343 V=10.0  +MOVJ EC344
SMOVL C344 V=10.0  +MOVJ EC345
SMOVL C345 V=10.0  +MOVJ EC346
SMOVL C346 V=10.0  +MOVJ EC347
SMOVL C347 V=10.0  +MOVJ EC348
SMOVL C348 V=10.0  +MOVJ EC349
SMOVL C349 V=10.0  +MOVJ EC350
SMOVL C350 V=10.0  +MOVJ EC351
SMOVL C351 V=10.0  +MOVJ EC352
WVOF
MACRO1 MJ#(10)
'LAYER_28
SMOVL C352 V=30.0  +MOVJ EC353
MACRO1 MJ#(16)
MACRO1 MJ#(9) ARGF30 ARGF0
WVON AMP=3.1 FREQ=2.5 ANGL=0.0 DIR=0
SMOVL C353 V=10.0  +MOVJ EC354
SMOVL C354 V=10.0  +MOVJ EC355
SMOVL C355 V=10.0  +MOVJ EC356
SMOVL C356 V=10.0  +MOVJ EC357
SMOVL C357 V=10.0  +MOVJ EC358
SMOVL C358 V=10.0  +MOVJ EC359
SMOVL C359 V=10.0  +MOVJ EC360
SMOVL C360 V=10.0  +MOVJ EC361
SMOVL C361 V=10.0  +MOVJ EC362
SMOVL C362 V=10.0  +MOVJ EC363
SMOVL C363 V=10.0  +MOVJ EC364
SMOVL C364 V=10.0  +MOVJ EC365
WVOF
MACRO1 MJ#(10)
'LAYER_29
SMOVL C365 V=30.0  +MOVJ EC366
MACRO1 MJ#(16)
MACRO1 MJ#(9) ARGF30 ARGF0
WVON AMP=3.1 FREQ=2.5 ANGL=0.0 DIR=0
SMOVL C366 V=10.0  +MOVJ EC367
SMOVL C367 V=10.0  +MOVJ EC368
SMOVL C368 V=10.0  +MOVJ EC369
SMOVL C369 V=10.0  +MOVJ EC370
SMOVL C370 V=10.0  +MOVJ EC371
SMOVL C371 V=10.0  +MOVJ EC372
SMOVL C372 V=10.0  +MOVJ EC373
SMOVL C373 V=10.0  +MOVJ EC374
SMOVL C374 V=10.0  +MOVJ EC375
SMOVL C375 V=10.0  +MOVJ EC376
SMOVL C376 V=10.0  +MOVJ EC377
SMOVL C377 V=10.0  +MOVJ EC378
WVOF
MACRO1 MJ#(10)
'LAYER_30
SMOVL C378 V=30.0  +MOVJ EC379
MACRO1 MJ#(16)
MACRO1 MJ#(9) ARGF30 ARGF0
WVON AMP=3.1 FREQ=2.5 ANGL=0.0 DIR=0
SMOVL C379 V=10.0  +MOVJ EC380
SMOVL C380 V=10.0  +MOVJ EC381
SMOVL C381 V=10.0  +MOVJ EC382
SMOVL C382 V=10.0  +MOVJ EC383
SMOVL C383 V=10.0  +MOVJ EC384
SMOVL C384 V=10.0  +MOVJ EC385
SMOVL C385 V=10.0  +MOVJ EC386
SMOVL C386 V=10.0  +MOVJ EC387
SMOVL C387 V=10.0  +MOVJ EC388
SMOVL C388 V=10.0  +MOVJ EC389
SMOVL C389 V=10.0  +MOVJ EC390
SMOVL C390 V=10.0  +MOVJ EC391
WVOF
MACRO1 MJ#(10)
'LAYER_31
SMOVL C391 V=30.0  +MOVJ EC392
MACRO1 MJ#(16)
MACRO1 MJ#(9) ARGF30 ARGF0
WVON AMP=3.1 FREQ=2.5 ANGL=0.0 DIR=0
SMOVL C392 V=10.0  +MOVJ EC393
SMOVL C393 V=10.0  +MOVJ EC394
SMOVL C394 V=10.0  +MOVJ EC395
SMOVL C395 V=10.0  +MOVJ EC396
SMOVL C396 V=10.0  +MOVJ EC397
SMOVL C397 V=10.0  +MOVJ EC398
SMOVL C398 V=10.0  +MOVJ EC399
SMOVL C399 V=10.0  +MOVJ EC400
SMOVL C400 V=10.0  +MOVJ EC401
SMOVL C401 V=10.0  +MOVJ EC402
SMOVL C402 V=10.0  +MOVJ EC403
SMOVL C403 V=10.0  +MOVJ EC404
WVOF
MACRO1 MJ#(10)
'LAYER_32
SMOVL C404 V=30.0  +MOVJ EC405
MACRO1 MJ#(16)
MACRO1 MJ#(9) ARGF30 ARGF0
WVON AMP=3.1 FREQ=2.5 ANGL=0.0 DIR=0
SMOVL C405 V=10.0  +MOVJ EC406
SMOVL C406 V=10.0  +MOVJ EC407
SMOVL C407 V=10.0  +MOVJ EC408
SMOVL C408 V=10.0  +MOVJ EC409
SMOVL C409 V=10.0  +MOVJ EC410
SMOVL C410 V=10.0  +MOVJ EC411
SMOVL C411 V=10.0  +MOVJ EC412
SMOVL C412 V=10.0  +MOVJ EC413
SMOVL C413 V=10.0  +MOVJ EC414
SMOVL C414 V=10.0  +MOVJ EC415
SMOVL C415 V=10.0  +MOVJ EC416
SMOVL C416 V=10.0  +MOVJ EC417
WVOF
MACRO1 MJ#(10)
'LAYER_33
SMOVL C417 V=30.0  +MOVJ EC418
MACRO1 MJ#(16)
MACRO1 MJ#(9) ARGF30 ARGF0
WVON AMP=3.1 FREQ=2.5 ANGL=0.0 DIR=0
SMOVL C418 V=10.0  +MOVJ EC419
SMOVL C419 V=10.0  +MOVJ EC420
SMOVL C420 V=10.0  +MOVJ EC421
SMOVL C421 V=10.0  +MOVJ EC422
SMOVL C422 V=10.0  +MOVJ EC423
SMOVL C423 V=10.0  +MOVJ EC424
SMOVL C424 V=10.0  +MOVJ EC425
SMOVL C425 V=10.0  +MOVJ EC426
SMOVL C426 V=10.0  +MOVJ EC427
SMOVL C427 V=10.0  +MOVJ EC428
SMOVL C428 V=10.0  +MOVJ EC429
SMOVL C429 V=10.0  +MOVJ EC430
WVOF
MACRO1 MJ#(10)
'LAYER_34
SMOVL C430 V=30.0  +MOVJ EC431
MACRO1 MJ#(16)
MACRO1 MJ#(9) ARGF30 ARGF0
WVON AMP=3.1 FREQ=2.5 ANGL=0.0 DIR=0
SMOVL C431 V=10.0  +MOVJ EC432
SMOVL C432 V=10.0  +MOVJ EC433
SMOVL C433 V=10.0  +MOVJ EC434
SMOVL C434 V=10.0  +MOVJ EC435
SMOVL C435 V=10.0  +MOVJ EC436
SMOVL C436 V=10.0  +MOVJ EC437
SMOVL C437 V=10.0  +MOVJ EC438
SMOVL C438 V=10.0  +MOVJ EC439
SMOVL C439 V=10.0  +MOVJ EC440
SMOVL C440 V=10.0  +MOVJ EC441
SMOVL C441 V=10.0  +MOVJ EC442
SMOVL C442 V=10.0  +MOVJ EC443
WVOF
MACRO1 MJ#(10)
'LAYER_35
SMOVL C443 V=30.0  +MOVJ EC444
MACRO1 MJ#(16)
MACRO1 MJ#(9) ARGF30 ARGF0
WVON AMP=3.1 FREQ=2.5 ANGL=0.0 DIR=0
SMOVL C444 V=10.0  +MOVJ EC445
SMOVL C445 V=10.0  +MOVJ EC446
SMOVL C446 V=10.0  +MOVJ EC447
SMOVL C447 V=10.0  +MOVJ EC448
SMOVL C448 V=10.0  +MOVJ EC449
SMOVL C449 V=10.0  +MOVJ EC450
SMOVL C450 V=10.0  +MOVJ EC451
SMOVL C451 V=10.0  +MOVJ EC452
SMOVL C452 V=10.0  +MOVJ EC453
SMOVL C453 V=10.0  +MOVJ EC454
SMOVL C454 V=10.0  +MOVJ EC455
SMOVL C455 V=10.0  +MOVJ EC456
WVOF
MACRO1 MJ#(10)
'LAYER_36
SMOVL C456 V=30.0  +MOVJ EC457
MACRO1 MJ#(16)
MACRO1 MJ#(9) ARGF30 ARGF0
WVON AMP=3.1 FREQ=2.5 ANGL=0.0 DIR=0
SMOVL C457 V=10.0  +MOVJ EC458
SMOVL C458 V=10.0  +MOVJ EC459
SMOVL C459 V=10.0  +MOVJ EC460
SMOVL C460 V=10.0  +MOVJ EC461
SMOVL C461 V=10.0  +MOVJ EC462
SMOVL C462 V=10.0  +MOVJ EC463
SMOVL C463 V=10.0  +MOVJ EC464
SMOVL C464 V=10.0  +MOVJ EC465
SMOVL C465 V=10.0  +MOVJ EC466
SMOVL C466 V=10.0  +MOVJ EC467
SMOVL C467 V=10.0  +MOVJ EC468
SMOVL C468 V=10.0  +MOVJ EC469
WVOF
MACRO1 MJ#(10)
'LAYER_37
SMOVL C469 V=30.0  +MOVJ EC470
MACRO1 MJ#(16)
MACRO1 MJ#(9) ARGF30 ARGF0
WVON AMP=3.1 FREQ=2.5 ANGL=0.0 DIR=0
SMOVL C470 V=10.0  +MOVJ EC471
SMOVL C471 V=10.0  +MOVJ EC472
SMOVL C472 V=10.0  +MOVJ EC473
SMOVL C473 V=10.0  +MOVJ EC474
SMOVL C474 V=10.0  +MOVJ EC475
SMOVL C475 V=10.0  +MOVJ EC476
SMOVL C476 V=10.0  +MOVJ EC477
SMOVL C477 V=10.0  +MOVJ EC478
SMOVL C478 V=10.0  +MOVJ EC479
SMOVL C479 V=10.0  +MOVJ EC480
SMOVL C480 V=10.0  +MOVJ EC481
SMOVL C481 V=10.0  +MOVJ EC482
WVOF
MACRO1 MJ#(10)
'LAYER_38
SMOVL C482 V=30.0  +MOVJ EC483
MACRO1 MJ#(16)
MACRO1 MJ#(9) ARGF30 ARGF0
WVON AMP=3.1 FREQ=2.5 ANGL=0.0 DIR=0
SMOVL C483 V=10.0  +MOVJ EC484
SMOVL C484 V=10.0  +MOVJ EC485
SMOVL C485 V=10.0  +MOVJ EC486
SMOVL C486 V=10.0  +MOVJ EC487
SMOVL C487 V=10.0  +MOVJ EC488
SMOVL C488 V=10.0  +MOVJ EC489
SMOVL C489 V=10.0  +MOVJ EC490
SMOVL C490 V=10.0  +MOVJ EC491
SMOVL C491 V=10.0  +MOVJ EC492
SMOVL C492 V=10.0  +MOVJ EC493
SMOVL C493 V=10.0  +MOVJ EC494
SMOVL C494 V=10.0  +MOVJ EC495
WVOF
MACRO1 MJ#(10)
'LAYER_39
SMOVL C495 V=30.0  +MOVJ EC496
MACRO1 MJ#(16)
MACRO1 MJ#(9) ARGF30 ARGF0
WVON AMP=3.1 FREQ=2.5 ANGL=0.0 DIR=0
SMOVL C496 V=10.0  +MOVJ EC497
SMOVL C497 V=10.0  +MOVJ EC498
SMOVL C498 V=10.0  +MOVJ EC499
SMOVL C499 V=10.0  +MOVJ EC500
SMOVL C500 V=10.0  +MOVJ EC501
SMOVL C501 V=10.0  +MOVJ EC502
SMOVL C502 V=10.0  +MOVJ EC503
SMOVL C503 V=10.0  +MOVJ EC504
SMOVL C504 V=10.0  +MOVJ EC505
SMOVL C505 V=10.0  +MOVJ EC506
SMOVL C506 V=10.0  +MOVJ EC507
SMOVL C507 V=10.0  +MOVJ EC508
WVOF
MACRO1 MJ#(10)
'LAYER_40
SMOVL C508 V=30.0  +MOVJ EC509
MACRO1 MJ#(16)
MACRO1 MJ#(9) ARGF30 ARGF0
WVON AMP=3.1 FREQ=2.5 ANGL=0.0 DIR=0
SMOVL C509 V=10.0  +MOVJ EC510
SMOVL C510 V=10.0  +MOVJ EC511
SMOVL C511 V=10.0  +MOVJ EC512
SMOVL C512 V=10.0  +MOVJ EC513
SMOVL C513 V=10.0  +MOVJ EC514
SMOVL C514 V=10.0  +MOVJ EC515
SMOVL C515 V=10.0  +MOVJ EC516
SMOVL C516 V=10.0  +MOVJ EC517
SMOVL C517 V=10.0  +MOVJ EC518
SMOVL C518 V=10.0  +MOVJ EC519
SMOVL C519 V=10.0  +MOVJ EC520
SMOVL C520 V=10.0  +MOVJ EC521
WVOF
MACRO1 MJ#(10)
'LAYER_41
SMOVL C521 V=30.0  +MOVJ EC522
MACRO1 MJ#(16)
MACRO1 MJ#(9) ARGF30 ARGF0
WVON AMP=3.1 FREQ=2.5 ANGL=0.0 DIR=0
SMOVL C522 V=10.0  +MOVJ EC523
SMOVL C523 V=10.0  +MOVJ EC524
SMOVL C524 V=10.0  +MOVJ EC525
SMOVL C525 V=10.0  +MOVJ EC526
SMOVL C526 V=10.0  +MOVJ EC527
SMOVL C527 V=10.0  +MOVJ EC528
SMOVL C528 V=10.0  +MOVJ EC529
SMOVL C529 V=10.0  +MOVJ EC530
SMOVL C530 V=10.0  +MOVJ EC531
SMOVL C531 V=10.0  +MOVJ EC532
SMOVL C532 V=10.0  +MOVJ EC533
SMOVL C533 V=10.0  +MOVJ EC534
WVOF
MACRO1 MJ#(10)
'LAYER_42
SMOVL C534 V=30.0  +MOVJ EC535
MACRO1 MJ#(16)
MACRO1 MJ#(9) ARGF30 ARGF0
WVON AMP=3.1 FREQ=2.5 ANGL=0.0 DIR=0
SMOVL C535 V=10.0  +MOVJ EC536
SMOVL C536 V=10.0  +MOVJ EC537
SMOVL C537 V=10.0  +MOVJ EC538
SMOVL C538 V=10.0  +MOVJ EC539
SMOVL C539 V=10.0  +MOVJ EC540
SMOVL C540 V=10.0  +MOVJ EC541
SMOVL C541 V=10.0  +MOVJ EC542
SMOVL C542 V=10.0  +MOVJ EC543
SMOVL C543 V=10.0  +MOVJ EC544
SMOVL C544 V=10.0  +MOVJ EC545
SMOVL C545 V=10.0  +MOVJ EC546
SMOVL C546 V=10.0  +MOVJ EC547
WVOF
MACRO1 MJ#(10)
'LAYER_43
SMOVL C547 V=30.0  +MOVJ EC548
MACRO1 MJ#(16)
MACRO1 MJ#(9) ARGF30 ARGF0
WVON AMP=3.1 FREQ=2.5 ANGL=0.0 DIR=0
SMOVL C548 V=10.0  +MOVJ EC549
SMOVL C549 V=10.0  +MOVJ EC550
SMOVL C550 V=10.0  +MOVJ EC551
SMOVL C551 V=10.0  +MOVJ EC552
SMOVL C552 V=10.0  +MOVJ EC553
SMOVL C553 V=10.0  +MOVJ EC554
SMOVL C554 V=10.0  +MOVJ EC555
SMOVL C555 V=10.0  +MOVJ EC556
SMOVL C556 V=10.0  +MOVJ EC557
SMOVL C557 V=10.0  +MOVJ EC558
SMOVL C558 V=10.0  +MOVJ EC559
SMOVL C559 V=10.0  +MOVJ EC560
WVOF
MACRO1 MJ#(10)
'LAYER_44
SMOVL C560 V=30.0  +MOVJ EC561
MACRO1 MJ#(16)
MACRO1 MJ#(9) ARGF30 ARGF0
WVON AMP=3.1 FREQ=2.5 ANGL=0.0 DIR=0
SMOVL C561 V=10.0  +MOVJ EC562
SMOVL C562 V=10.0  +MOVJ EC563
SMOVL C563 V=10.0  +MOVJ EC564
SMOVL C564 V=10.0  +MOVJ EC565
SMOVL C565 V=10.0  +MOVJ EC566
SMOVL C566 V=10.0  +MOVJ EC567
SMOVL C567 V=10.0  +MOVJ EC568
SMOVL C568 V=10.0  +MOVJ EC569
SMOVL C569 V=10.0  +MOVJ EC570
SMOVL C570 V=10.0  +MOVJ EC571
SMOVL C571 V=10.0  +MOVJ EC572
SMOVL C572 V=10.0  +MOVJ EC573
WVOF
MACRO1 MJ#(10)
'LAYER_45
SMOVL C573 V=30.0  +MOVJ EC574
MACRO1 MJ#(16)
MACRO1 MJ#(9) ARGF30 ARGF0
WVON AMP=3.1 FREQ=2.5 ANGL=0.0 DIR=0
SMOVL C574 V=10.0  +MOVJ EC575
SMOVL C575 V=10.0  +MOVJ EC576
SMOVL C576 V=10.0  +MOVJ EC577
SMOVL C577 V=10.0  +MOVJ EC578
SMOVL C578 V=10.0  +MOVJ EC579
SMOVL C579 V=10.0  +MOVJ EC580
SMOVL C580 V=10.0  +MOVJ EC581
SMOVL C581 V=10.0  +MOVJ EC582
SMOVL C582 V=10.0  +MOVJ EC583
SMOVL C583 V=10.0  +MOVJ EC584
SMOVL C584 V=10.0  +MOVJ EC585
SMOVL C585 V=10.0  +MOVJ EC586
WVOF
MACRO1 MJ#(10)
'LAYER_46
SMOVL C586 V=30.0  +MOVJ EC587
MACRO1 MJ#(16)
MACRO1 MJ#(9) ARGF30 ARGF0
WVON AMP=3.1 FREQ=2.5 ANGL=0.0 DIR=0
SMOVL C587 V=10.0  +MOVJ EC588
SMOVL C588 V=10.0  +MOVJ EC589
SMOVL C589 V=10.0  +MOVJ EC590
SMOVL C590 V=10.0  +MOVJ EC591
SMOVL C591 V=10.0  +MOVJ EC592
SMOVL C592 V=10.0  +MOVJ EC593
SMOVL C593 V=10.0  +MOVJ EC594
SMOVL C594 V=10.0  +MOVJ EC595
SMOVL C595 V=10.0  +MOVJ EC596
SMOVL C596 V=10.0  +MOVJ EC597
SMOVL C597 V=10.0  +MOVJ EC598
SMOVL C598 V=10.0  +MOVJ EC599
WVOF
MACRO1 MJ#(10)
'LAYER_47
SMOVL C599 V=30.0  +MOVJ EC600
MACRO1 MJ#(16)
MACRO1 MJ#(9) ARGF30 ARGF0
WVON AMP=3.1 FREQ=2.5 ANGL=0.0 DIR=0
SMOVL C600 V=10.0  +MOVJ EC601
SMOVL C601 V=10.0  +MOVJ EC602
SMOVL C602 V=10.0  +MOVJ EC603
SMOVL C603 V=10.0  +MOVJ EC604
SMOVL C604 V=10.0  +MOVJ EC605
SMOVL C605 V=10.0  +MOVJ EC606
SMOVL C606 V=10.0  +MOVJ EC607
SMOVL C607 V=10.0  +MOVJ EC608
SMOVL C608 V=10.0  +MOVJ EC609
SMOVL C609 V=10.0  +MOVJ EC610
SMOVL C610 V=10.0  +MOVJ EC611
SMOVL C611 V=10.0  +MOVJ EC612
WVOF
MACRO1 MJ#(10)
'LAYER_48
SMOVL C612 V=30.0  +MOVJ EC613
MACRO1 MJ#(16)
MACRO1 MJ#(9) ARGF30 ARGF0
WVON AMP=3.1 FREQ=2.5 ANGL=0.0 DIR=0
SMOVL C613 V=10.0  +MOVJ EC614
SMOVL C614 V=10.0  +MOVJ EC615
SMOVL C615 V=10.0  +MOVJ EC616
SMOVL C616 V=10.0  +MOVJ EC617
SMOVL C617 V=10.0  +MOVJ EC618
SMOVL C618 V=10.0  +MOVJ EC619
SMOVL C619 V=10.0  +MOVJ EC620
SMOVL C620 V=10.0  +MOVJ EC621
SMOVL C621 V=10.0  +MOVJ EC622
SMOVL C622 V=10.0  +MOVJ EC623
SMOVL C623 V=10.0  +MOVJ EC624
SMOVL C624 V=10.0  +MOVJ EC625
WVOF
MACRO1 MJ#(10)
'LAYER_49
SMOVL C625 V=30.0  +MOVJ EC626
MACRO1 MJ#(16)
MACRO1 MJ#(9) ARGF30 ARGF0
WVON AMP=3.1 FREQ=2.5 ANGL=0.0 DIR=0
SMOVL C626 V=10.0  +MOVJ EC627
SMOVL C627 V=10.0  +MOVJ EC628
SMOVL C628 V=10.0  +MOVJ EC629
SMOVL C629 V=10.0  +MOVJ EC630
SMOVL C630 V=10.0  +MOVJ EC631
SMOVL C631 V=10.0  +MOVJ EC632
SMOVL C632 V=10.0  +MOVJ EC633
SMOVL C633 V=10.0  +MOVJ EC634
SMOVL C634 V=10.0  +MOVJ EC635
SMOVL C635 V=10.0  +MOVJ EC636
SMOVL C636 V=10.0  +MOVJ EC637
SMOVL C637 V=10.0  +MOVJ EC638
WVOF
MACRO1 MJ#(10)
END
